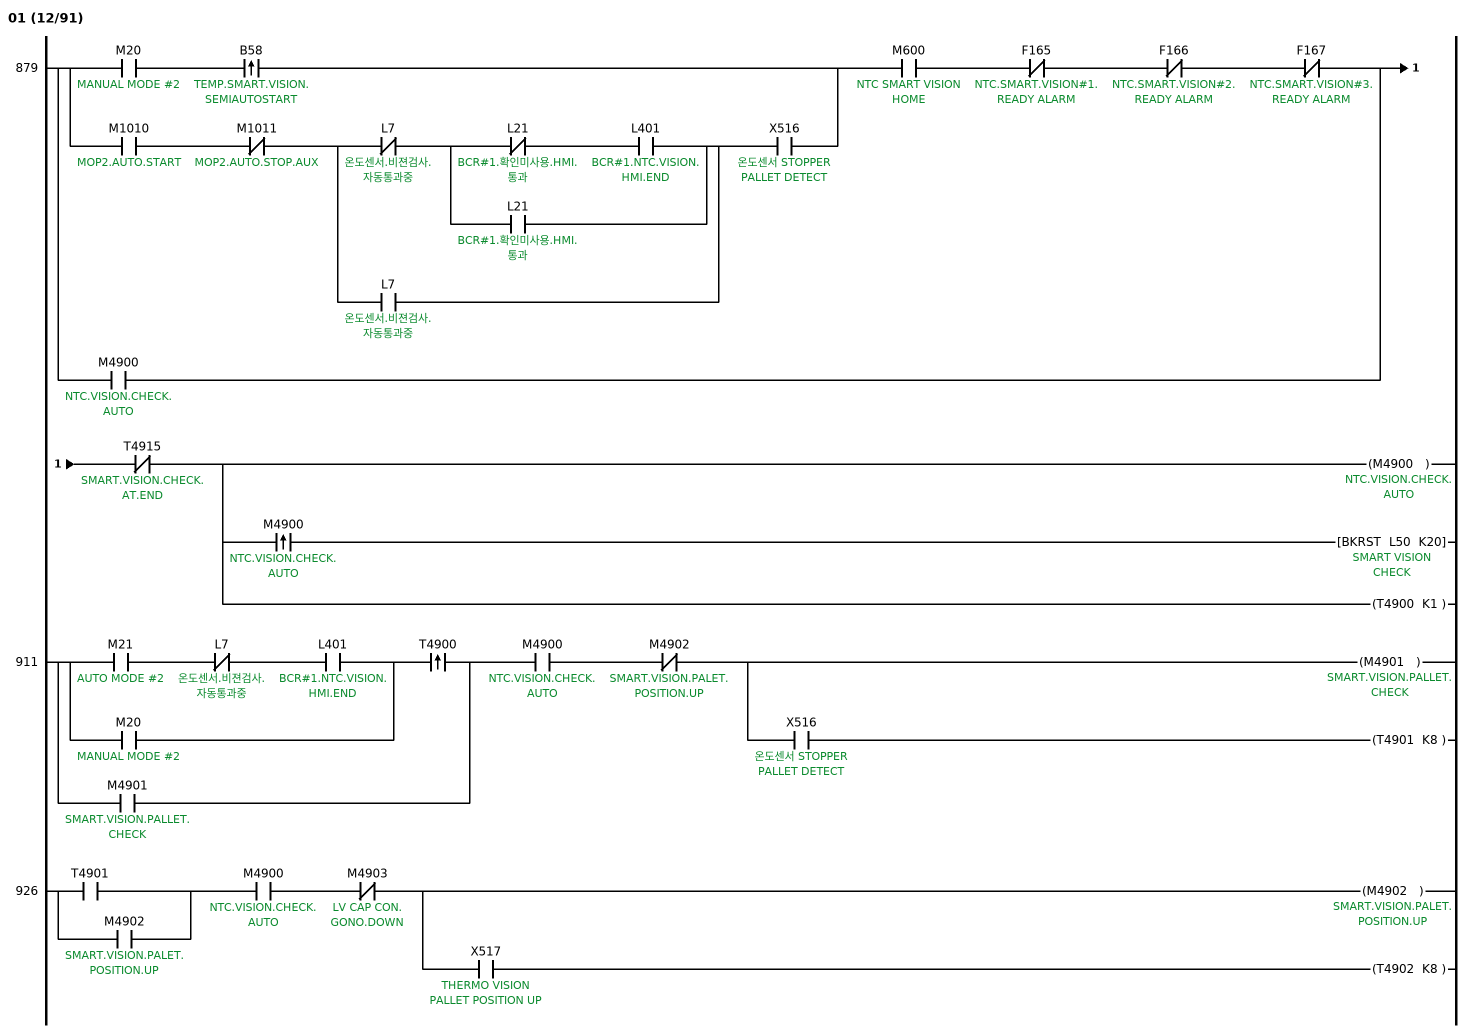
879   LD      M20  ; MANUAL MODE #2
      ANDP    B58  ; TEMP.SMART.VISION.SEMIAUTOSTART
      LD      M1010  ; MOP2.AUTO.START
      ANI     M1011  ; MOP2.AUTO.STOP.AUX
      LDI     L7  ; 온도센서.비젼검사.자동통과중
      LDI     L21  ; BCR#1.확인미사용.HMI.통과
      AND     L401  ; BCR#1.NTC.VISION.HMI.END
      OR      L21  ; BCR#1.확인미사용.HMI.통과
      ANB
      OR      L7  ; 온도센서.비젼검사.자동통과중
      ANB
      AND     X516  ; 온도센서 STOPPER PALLET DETECT
      ORB
      AND     M600  ; NTC SMART VISION HOME
      ANI     F165  ; NTC.SMART.VISION#1.READY ALARM
      ANI     F166  ; NTC.SMART.VISION#2.READY ALARM
      ANI     F167  ; NTC.SMART.VISION#3.READY ALARM
      OR      M4900  ; NTC.VISION.CHECK.AUTO
      ANI     T4915  ; SMART.VISION.CHECK.AT.END
      OUT     M4900  ; NTC.VISION.CHECK.AUTO
      MPS
      ANDP    M4900  ; NTC.VISION.CHECK.AUTO
      BKRST   L50 K20  ; SMART VISION CHECK
      MPP
      OUT     T4900 K1
911   LD      M21  ; AUTO MODE #2
      ANI     L7  ; 온도센서.비젼검사.자동통과중
      AND     L401  ; BCR#1.NTC.VISION.HMI.END
      OR      M20  ; MANUAL MODE #2
      ANDP    T4900
      OR      M4901  ; SMART.VISION.PALLET.CHECK
      AND     M4900  ; NTC.VISION.CHECK.AUTO
      ANI     M4902  ; SMART.VISION.PALET.POSITION.UP
      OUT     M4901  ; SMART.VISION.PALLET.CHECK
      AND     X516  ; 온도센서 STOPPER PALLET DETECT
      OUT     T4901 K8
926   LD      T4901
      OR      M4902  ; SMART.VISION.PALET.POSITION.UP
      AND     M4900  ; NTC.VISION.CHECK.AUTO
      ANI     M4903  ; LV CAP CON. GONO.DOWN
      OUT     M4902  ; SMART.VISION.PALET.POSITION.UP
      AND     X517  ; THERMO VISION PALLET POSITION UP
      OUT     T4902 K8
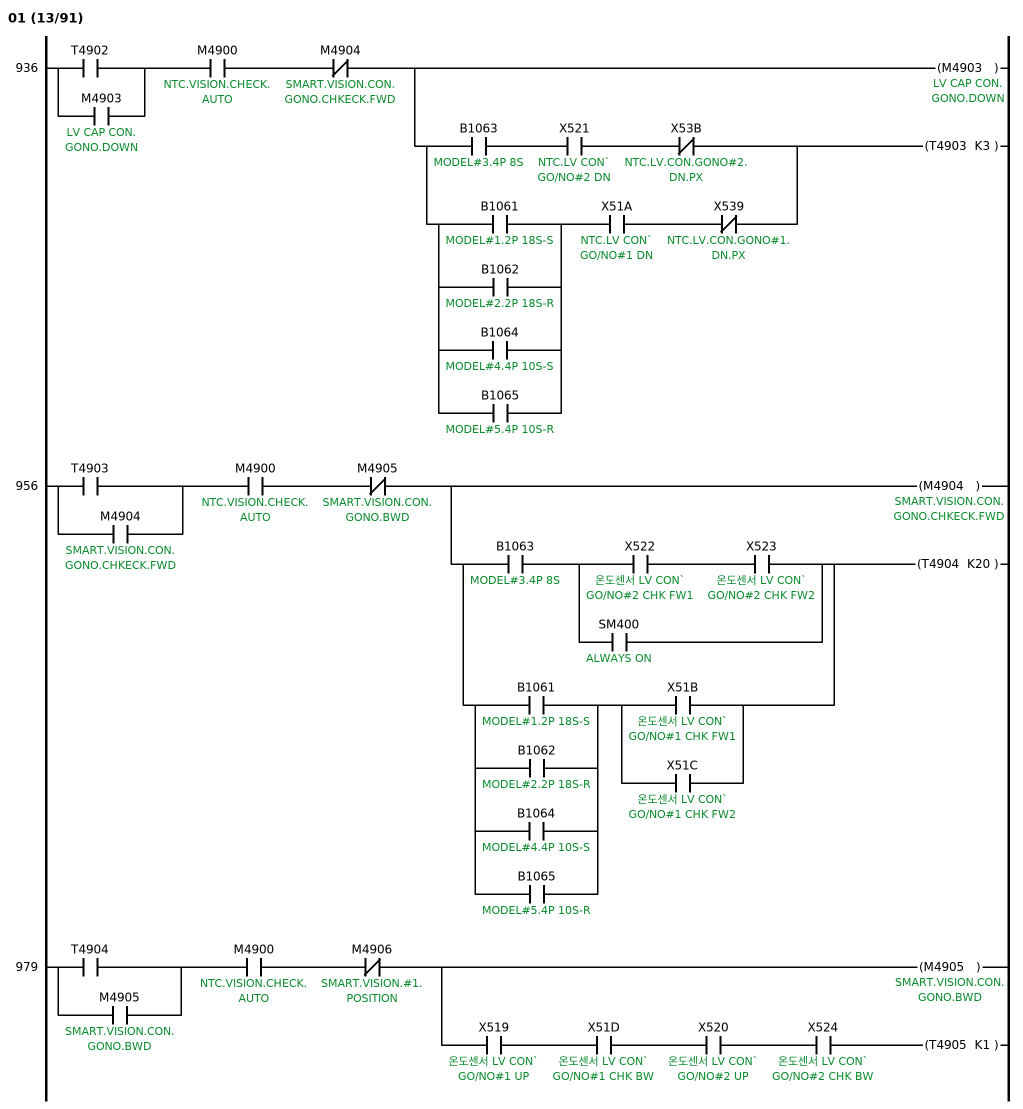
936   LD      T4902
      OR      M4903  ; LV CAP CON. GONO.DOWN
      AND     M4900  ; NTC.VISION.CHECK.AUTO
      ANI     M4904  ; SMART.VISION.CON.GONO.CHKECK.FWD
      OUT     M4903  ; LV CAP CON. GONO.DOWN
      LD      B1063  ; MODEL#3.4P 8S
      AND     X521  ; NTC.LV CON` GO/NO#2 DN
      ANI     X53B  ; NTC.LV.CON.GONO#2.DN.PX
      LD      B1061  ; MODEL#1.2P 18S-S
      OR      B1062  ; MODEL#2.2P 18S-R
      OR      B1064  ; MODEL#4.4P 10S-S
      OR      B1065  ; MODEL#5.4P 10S-R
      AND     X51A  ; NTC.LV CON` GO/NO#1 DN
      ANI     X539  ; NTC.LV.CON.GONO#1.DN.PX
      ORB
      ANB
      OUT     T4903 K3
956   LD      T4903
      OR      M4904  ; SMART.VISION.CON.GONO.CHKECK.FWD
      AND     M4900  ; NTC.VISION.CHECK.AUTO
      ANI     M4905  ; SMART.VISION.CON.GONO.BWD
      OUT     M4904  ; SMART.VISION.CON.GONO.CHKECK.FWD
      LD      B1063  ; MODEL#3.4P 8S
      LD      X522  ; 온도센서 LV CON` GO/NO#2 CHK FW1
      AND     X523  ; 온도센서 LV CON` GO/NO#2 CHK FW2
      OR      SM400  ; ALWAYS ON
      ANB
      LD      B1061  ; MODEL#1.2P 18S-S
      OR      B1062  ; MODEL#2.2P 18S-R
      OR      B1064  ; MODEL#4.4P 10S-S
      OR      B1065  ; MODEL#5.4P 10S-R
      LD      X51B  ; 온도센서 LV CON` GO/NO#1 CHK FW1
      OR      X51C  ; 온도센서 LV CON` GO/NO#1 CHK FW2
      ANB
      ORB
      ANB
      OUT     T4904 K20
979   LD      T4904
      OR      M4905  ; SMART.VISION.CON.GONO.BWD
      AND     M4900  ; NTC.VISION.CHECK.AUTO
      ANI     M4906  ; SMART.VISION.#1.POSITION
      OUT     M4905  ; SMART.VISION.CON.GONO.BWD
      AND     X519  ; 온도센서 LV CON` GO/NO#1 UP
      AND     X51D  ; 온도센서 LV CON` GO/NO#1 CHK BW
      AND     X520  ; 온도센서 LV CON` GO/NO#2 UP
      AND     X524  ; 온도센서 LV CON` GO/NO#2 CHK BW
      OUT     T4905 K1
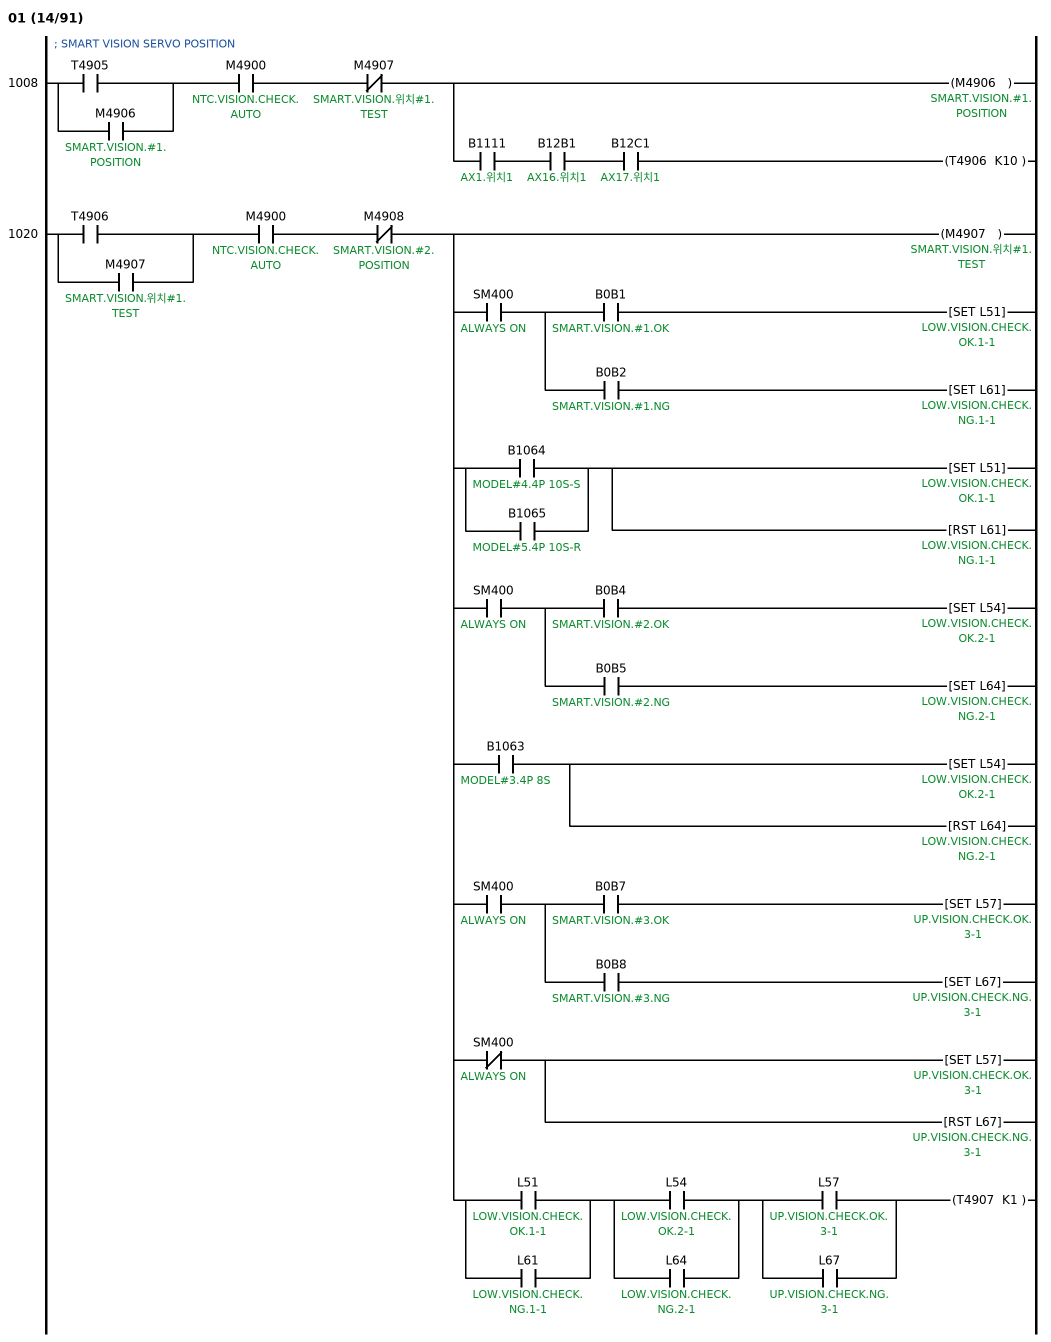
; SMART VISION SERVO POSITION
1008  LD      T4905
      OR      M4906  ; SMART.VISION.#1.POSITION
      AND     M4900  ; NTC.VISION.CHECK.AUTO
      ANI     M4907  ; SMART.VISION.위치#1.TEST
      OUT     M4906  ; SMART.VISION.#1.POSITION
      AND     B1111  ; AX1.위치1
      AND     B12B1  ; AX16.위치1
      AND     B12C1  ; AX17.위치1
      OUT     T4906 K10
1020  LD      T4906
      OR      M4907  ; SMART.VISION.위치#1.TEST
      AND     M4900  ; NTC.VISION.CHECK.AUTO
      ANI     M4908  ; SMART.VISION.#2.POSITION
      OUT     M4907  ; SMART.VISION.위치#1.TEST
      MPS
      AND     SM400  ; ALWAYS ON
      MPS
      AND     B0B1  ; SMART.VISION.#1.OK
      SET     L51  ; LOW.VISION.CHECK.OK.1-1
      MPP
      AND     B0B2  ; SMART.VISION.#1.NG
      SET     L61  ; LOW.VISION.CHECK.NG.1-1
      MRD
      LD      B1064  ; MODEL#4.4P 10S-S
      OR      B1065  ; MODEL#5.4P 10S-R
      ANB
      SET     L51  ; LOW.VISION.CHECK.OK.1-1
      RST     L61  ; LOW.VISION.CHECK.NG.1-1
      MRD
      AND     SM400  ; ALWAYS ON
      MPS
      AND     B0B4  ; SMART.VISION.#2.OK
      SET     L54  ; LOW.VISION.CHECK.OK.2-1
      MPP
      AND     B0B5  ; SMART.VISION.#2.NG
      SET     L64  ; LOW.VISION.CHECK.NG.2-1
      MRD
      AND     B1063  ; MODEL#3.4P 8S
      SET     L54  ; LOW.VISION.CHECK.OK.2-1
      RST     L64  ; LOW.VISION.CHECK.NG.2-1
      MRD
      AND     SM400  ; ALWAYS ON
      MPS
      AND     B0B7  ; SMART.VISION.#3.OK
      SET     L57  ; UP.VISION.CHECK.OK.3-1
      MPP
      AND     B0B8  ; SMART.VISION.#3.NG
      SET     L67  ; UP.VISION.CHECK.NG.3-1
      MRD
      ANI     SM400  ; ALWAYS ON
      SET     L57  ; UP.VISION.CHECK.OK.3-1
      RST     L67  ; UP.VISION.CHECK.NG.3-1
      MPP
      LD      L51  ; LOW.VISION.CHECK.OK.1-1
      OR      L61  ; LOW.VISION.CHECK.NG.1-1
      ANB
      LD      L54  ; LOW.VISION.CHECK.OK.2-1
      OR      L64  ; LOW.VISION.CHECK.NG.2-1
      ANB
      LD      L57  ; UP.VISION.CHECK.OK.3-1
      OR      L67  ; UP.VISION.CHECK.NG.3-1
      ANB
      OUT     T4907 K1
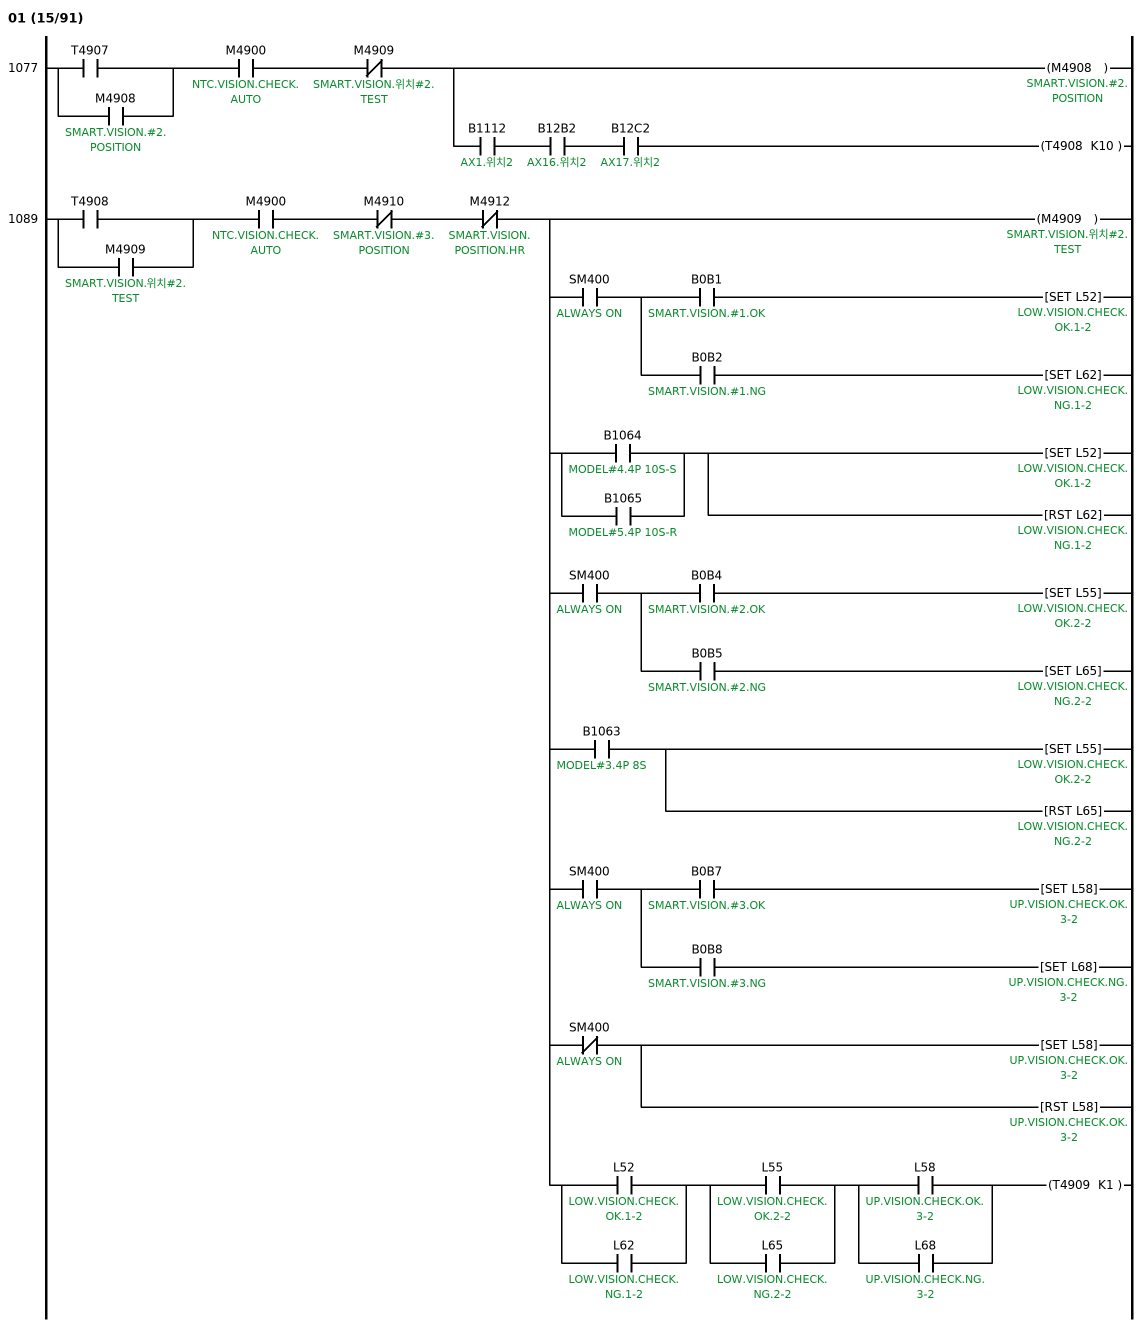
1077  LD      T4907
      OR      M4908  ; SMART.VISION.#2.POSITION
      AND     M4900  ; NTC.VISION.CHECK.AUTO
      ANI     M4909  ; SMART.VISION.위치#2.TEST
      OUT     M4908  ; SMART.VISION.#2.POSITION
      AND     B1112  ; AX1.위치2
      AND     B12B2  ; AX16.위치2
      AND     B12C2  ; AX17.위치2
      OUT     T4908 K10
1089  LD      T4908
      OR      M4909  ; SMART.VISION.위치#2.TEST
      AND     M4900  ; NTC.VISION.CHECK.AUTO
      ANI     M4910  ; SMART.VISION.#3.POSITION
      ANI     M4912  ; SMART.VISION.POSITION.HR
      OUT     M4909  ; SMART.VISION.위치#2.TEST
      MPS
      AND     SM400  ; ALWAYS ON
      MPS
      AND     B0B1  ; SMART.VISION.#1.OK
      SET     L52  ; LOW.VISION.CHECK.OK.1-2
      MPP
      AND     B0B2  ; SMART.VISION.#1.NG
      SET     L62  ; LOW.VISION.CHECK.NG.1-2
      MRD
      LD      B1064  ; MODEL#4.4P 10S-S
      OR      B1065  ; MODEL#5.4P 10S-R
      ANB
      SET     L52  ; LOW.VISION.CHECK.OK.1-2
      RST     L62  ; LOW.VISION.CHECK.NG.1-2
      MRD
      AND     SM400  ; ALWAYS ON
      MPS
      AND     B0B4  ; SMART.VISION.#2.OK
      SET     L55  ; LOW.VISION.CHECK.OK.2-2
      MPP
      AND     B0B5  ; SMART.VISION.#2.NG
      SET     L65  ; LOW.VISION.CHECK.NG.2-2
      MRD
      AND     B1063  ; MODEL#3.4P 8S
      SET     L55  ; LOW.VISION.CHECK.OK.2-2
      RST     L65  ; LOW.VISION.CHECK.NG.2-2
      MRD
      AND     SM400  ; ALWAYS ON
      MPS
      AND     B0B7  ; SMART.VISION.#3.OK
      SET     L58  ; UP.VISION.CHECK.OK.3-2
      MPP
      AND     B0B8  ; SMART.VISION.#3.NG
      SET     L68  ; UP.VISION.CHECK.NG.3-2
      MRD
      ANI     SM400  ; ALWAYS ON
      SET     L58  ; UP.VISION.CHECK.OK.3-2
      RST     L58  ; UP.VISION.CHECK.OK.3-2
      MPP
      LD      L52  ; LOW.VISION.CHECK.OK.1-2
      OR      L62  ; LOW.VISION.CHECK.NG.1-2
      ANB
      LD      L55  ; LOW.VISION.CHECK.OK.2-2
      OR      L65  ; LOW.VISION.CHECK.NG.2-2
      ANB
      LD      L58  ; UP.VISION.CHECK.OK.3-2
      OR      L68  ; UP.VISION.CHECK.NG.3-2
      ANB
      OUT     T4909 K1
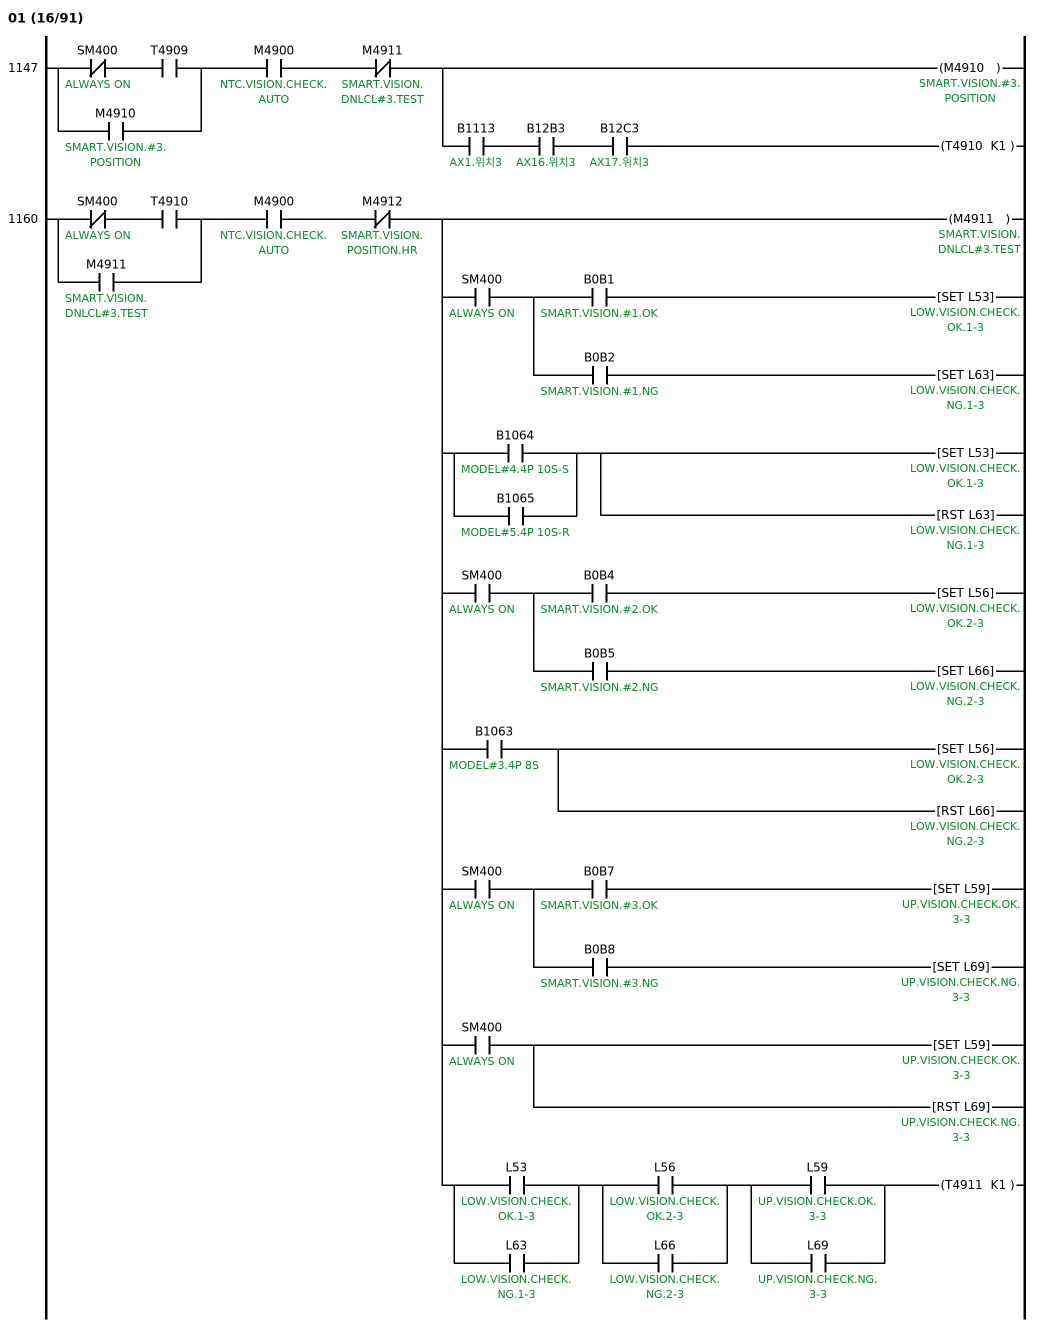
1147  LDI     SM400  ; ALWAYS ON
      AND     T4909
      OR      M4910  ; SMART.VISION.#3.POSITION
      AND     M4900  ; NTC.VISION.CHECK.AUTO
      ANI     M4911  ; SMART.VISION.DNLCL#3.TEST
      OUT     M4910  ; SMART.VISION.#3.POSITION
      AND     B1113  ; AX1.위치3
      AND     B12B3  ; AX16.위치3
      AND     B12C3  ; AX17.위치3
      OUT     T4910 K1
1160  LDI     SM400  ; ALWAYS ON
      AND     T4910
      OR      M4911  ; SMART.VISION.DNLCL#3.TEST
      AND     M4900  ; NTC.VISION.CHECK.AUTO
      ANI     M4912  ; SMART.VISION.POSITION.HR
      OUT     M4911  ; SMART.VISION.DNLCL#3.TEST
      MPS
      AND     SM400  ; ALWAYS ON
      MPS
      AND     B0B1  ; SMART.VISION.#1.OK
      SET     L53  ; LOW.VISION.CHECK.OK.1-3
      MPP
      AND     B0B2  ; SMART.VISION.#1.NG
      SET     L63  ; LOW.VISION.CHECK.NG.1-3
      MRD
      LD      B1064  ; MODEL#4.4P 10S-S
      OR      B1065  ; MODEL#5.4P 10S-R
      ANB
      SET     L53  ; LOW.VISION.CHECK.OK.1-3
      RST     L63  ; LOW.VISION.CHECK.NG.1-3
      MRD
      AND     SM400  ; ALWAYS ON
      MPS
      AND     B0B4  ; SMART.VISION.#2.OK
      SET     L56  ; LOW.VISION.CHECK.OK.2-3
      MPP
      AND     B0B5  ; SMART.VISION.#2.NG
      SET     L66  ; LOW.VISION.CHECK.NG.2-3
      MRD
      AND     B1063  ; MODEL#3.4P 8S
      SET     L56  ; LOW.VISION.CHECK.OK.2-3
      RST     L66  ; LOW.VISION.CHECK.NG.2-3
      MRD
      AND     SM400  ; ALWAYS ON
      MPS
      AND     B0B7  ; SMART.VISION.#3.OK
      SET     L59  ; UP.VISION.CHECK.OK.3-3
      MPP
      AND     B0B8  ; SMART.VISION.#3.NG
      SET     L69  ; UP.VISION.CHECK.NG.3-3
      MRD
      AND     SM400  ; ALWAYS ON
      SET     L59  ; UP.VISION.CHECK.OK.3-3
      RST     L69  ; UP.VISION.CHECK.NG.3-3
      MPP
      LD      L53  ; LOW.VISION.CHECK.OK.1-3
      OR      L63  ; LOW.VISION.CHECK.NG.1-3
      ANB
      LD      L56  ; LOW.VISION.CHECK.OK.2-3
      OR      L66  ; LOW.VISION.CHECK.NG.2-3
      ANB
      LD      L59  ; UP.VISION.CHECK.OK.3-3
      OR      L69  ; UP.VISION.CHECK.NG.3-3
      ANB
      OUT     T4911 K1
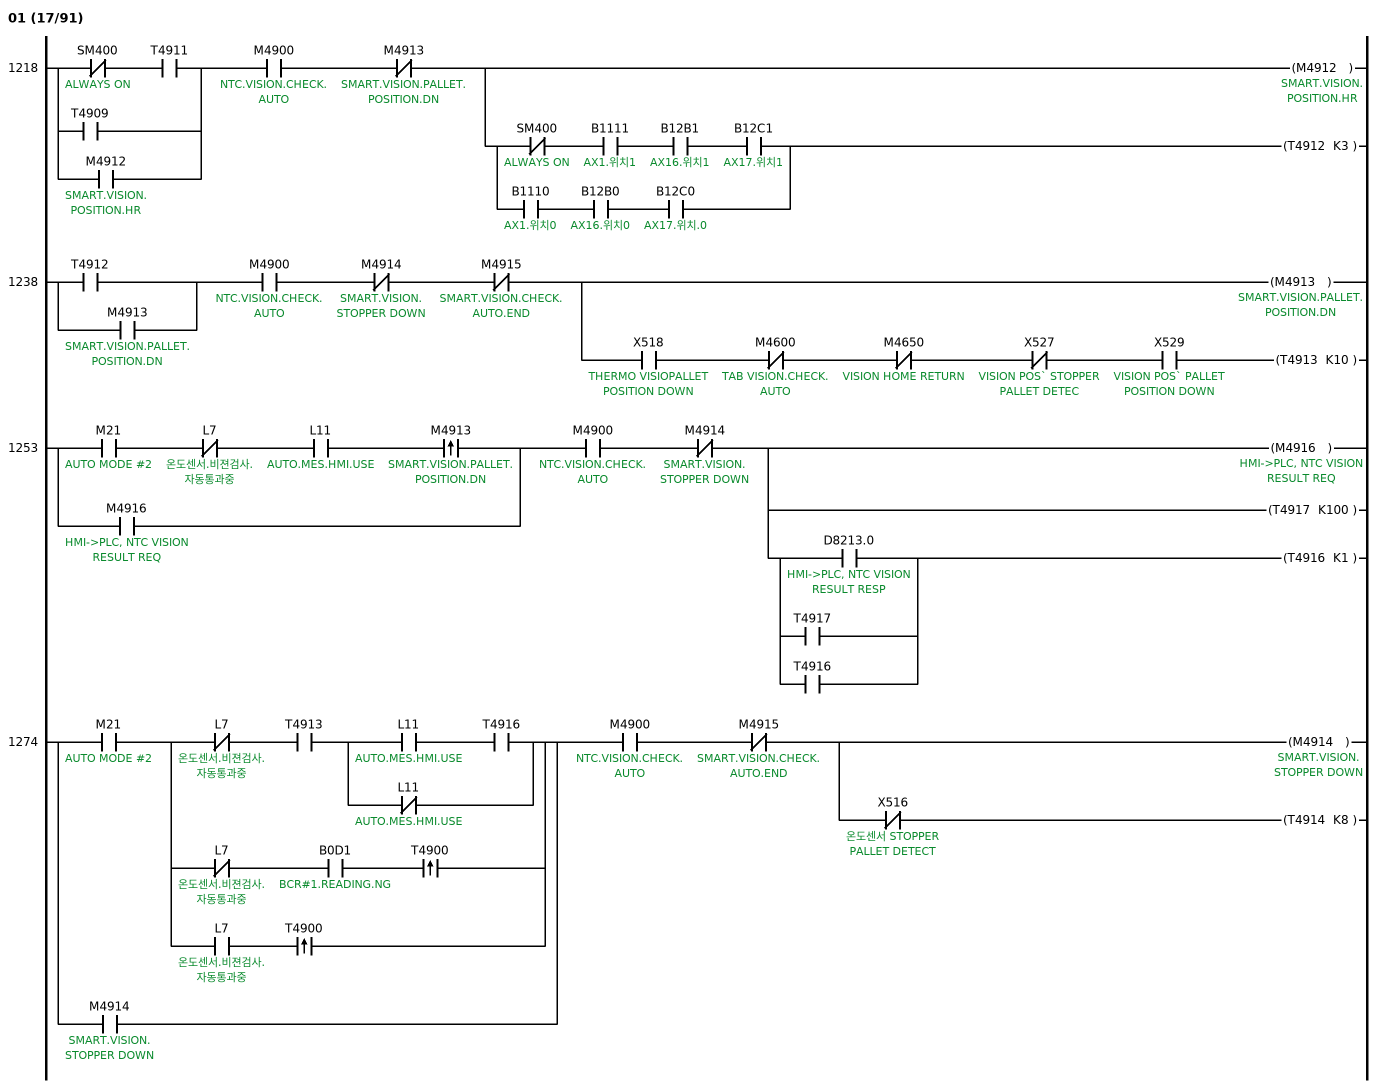
1218  LDI     SM400  ; ALWAYS ON
      AND     T4911
      OR      T4909
      OR      M4912  ; SMART.VISION.POSITION.HR
      AND     M4900  ; NTC.VISION.CHECK.AUTO
      ANI     M4913  ; SMART.VISION.PALLET.POSITION.DN
      OUT     M4912  ; SMART.VISION.POSITION.HR
      LDI     SM400  ; ALWAYS ON
      AND     B1111  ; AX1.위치1
      AND     B12B1  ; AX16.위치1
      AND     B12C1  ; AX17.위치1
      LD      B1110  ; AX1.위치0
      AND     B12B0  ; AX16.위치0
      AND     B12C0  ; AX17.위치.0
      ORB
      ANB
      OUT     T4912 K3
1238  LD      T4912
      OR      M4913  ; SMART.VISION.PALLET.POSITION.DN
      AND     M4900  ; NTC.VISION.CHECK.AUTO
      ANI     M4914  ; SMART.VISION.STOPPER DOWN
      ANI     M4915  ; SMART.VISION.CHECK.AUTO.END
      OUT     M4913  ; SMART.VISION.PALLET.POSITION.DN
      AND     X518  ; THERMO VISIOPALLET POSITION DOWN
      ANI     M4600  ; TAB VISION.CHECK.AUTO
      ANI     M4650  ; VISION HOME RETURN
      ANI     X527  ; VISION POS` STOPPER PALLET DETEC
      AND     X529  ; VISION POS` PALLET POSITION DOWN
      OUT     T4913 K10
1253  LD      M21  ; AUTO MODE #2
      ANI     L7  ; 온도센서.비젼검사.자동통과중
      AND     L11  ; AUTO.MES.HMI.USE
      ANDP    M4913  ; SMART.VISION.PALLET.POSITION.DN
      OR      M4916  ; HMI->PLC, NTC VISION RESULT REQ
      AND     M4900  ; NTC.VISION.CHECK.AUTO
      ANI     M4914  ; SMART.VISION.STOPPER DOWN
      OUT     M4916  ; HMI->PLC, NTC VISION RESULT REQ
      OUT     T4917 K100
      LD      D8213.0  ; HMI->PLC, NTC VISION RESULT RESP
      OR      T4917
      OR      T4916
      ANB
      OUT     T4916 K1
1274  LD      M21  ; AUTO MODE #2
      LDI     L7  ; 온도센서.비젼검사.자동통과중
      AND     T4913
      LD      L11  ; AUTO.MES.HMI.USE
      AND     T4916
      ORI     L11  ; AUTO.MES.HMI.USE
      ANB
      LDI     L7  ; 온도센서.비젼검사.자동통과중
      AND     B0D1  ; BCR#1.READING.NG
      ANDP    T4900
      ORB
      LD      L7  ; 온도센서.비젼검사.자동통과중
      ANDP    T4900
      ORB
      ANB
      OR      M4914  ; SMART.VISION.STOPPER DOWN
      AND     M4900  ; NTC.VISION.CHECK.AUTO
      ANI     M4915  ; SMART.VISION.CHECK.AUTO.END
      OUT     M4914  ; SMART.VISION.STOPPER DOWN
      ANI     X516  ; 온도센서 STOPPER PALLET DETECT
      OUT     T4914 K8
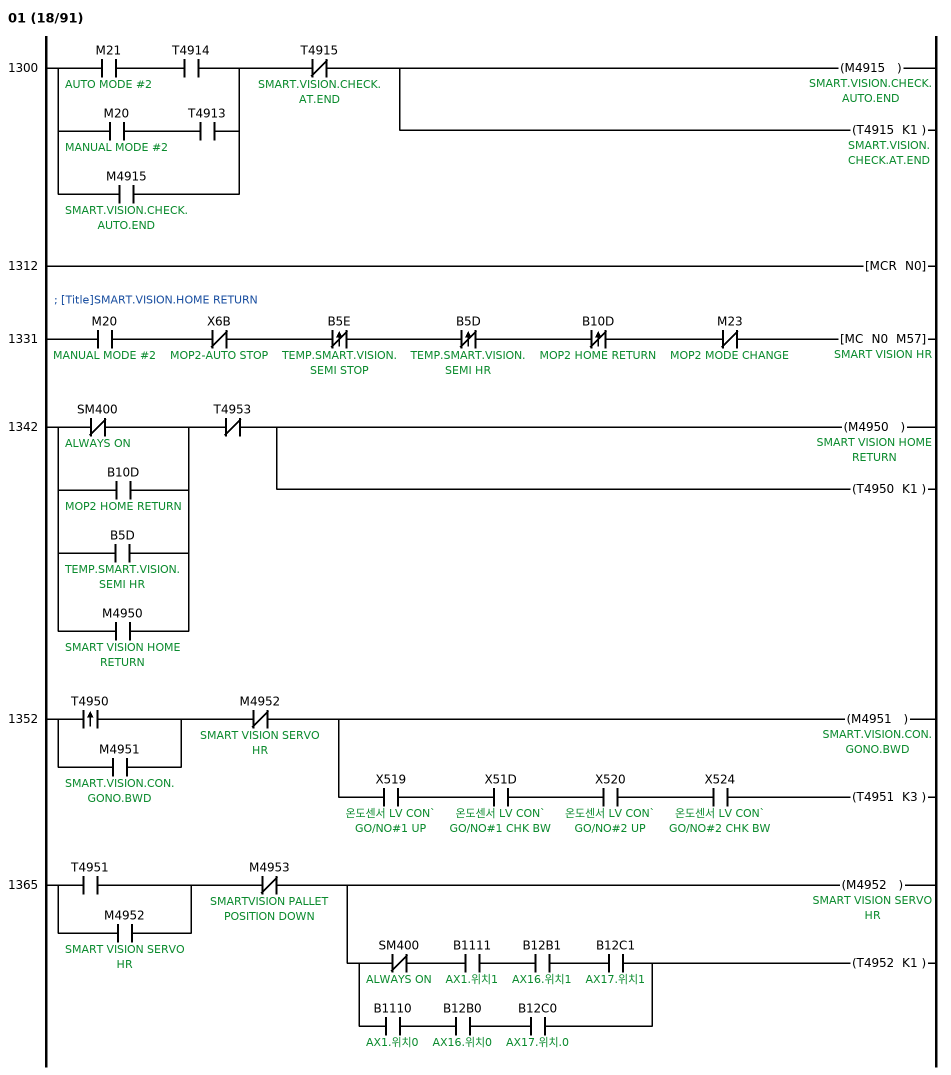
1300  LD      M21  ; AUTO MODE #2
      AND     T4914
      LD      M20  ; MANUAL MODE #2
      AND     T4913
      ORB
      OR      M4915  ; SMART.VISION.CHECK.AUTO.END
      ANI     T4915  ; SMART.VISION.CHECK.AT.END
      OUT     M4915  ; SMART.VISION.CHECK.AUTO.END
      OUT     T4915 K1  ; SMART.VISION.CHECK.AT.END
1312  MCR     N0
; [Title]SMART.VISION.HOME RETURN
1331  LD      M20  ; MANUAL MODE #2
      ANI     X6B  ; MOP2-AUTO STOP
      ANDPI   B5E  ; TEMP.SMART.VISION.SEMI STOP
      ANDPI   B5D  ; TEMP.SMART.VISION.SEMI HR
      ANDPI   B10D  ; MOP2 HOME RETURN
      ANI     M23  ; MOP2 MODE CHANGE
      MC      N0 M57  ; SMART VISION HR
1342  LDI     SM400  ; ALWAYS ON
      OR      B10D  ; MOP2 HOME RETURN
      OR      B5D  ; TEMP.SMART.VISION.SEMI HR
      OR      M4950  ; SMART VISION HOME RETURN
      ANI     T4953
      OUT     M4950  ; SMART VISION HOME RETURN
      OUT     T4950 K1
1352  LDP     T4950
      OR      M4951  ; SMART.VISION.CON.GONO.BWD
      ANI     M4952  ; SMART VISION SERVO HR
      OUT     M4951  ; SMART.VISION.CON.GONO.BWD
      AND     X519  ; 온도센서 LV CON` GO/NO#1 UP
      AND     X51D  ; 온도센서 LV CON` GO/NO#1 CHK BW
      AND     X520  ; 온도센서 LV CON` GO/NO#2 UP
      AND     X524  ; 온도센서 LV CON` GO/NO#2 CHK BW
      OUT     T4951 K3
1365  LD      T4951
      OR      M4952  ; SMART VISION SERVO HR
      ANI     M4953  ; SMARTVISION PALLET POSITION DOWN
      OUT     M4952  ; SMART VISION SERVO HR
      LDI     SM400  ; ALWAYS ON
      AND     B1111  ; AX1.위치1
      AND     B12B1  ; AX16.위치1
      AND     B12C1  ; AX17.위치1
      LD      B1110  ; AX1.위치0
      AND     B12B0  ; AX16.위치0
      AND     B12C0  ; AX17.위치.0
      ORB
      ANB
      OUT     T4952 K1
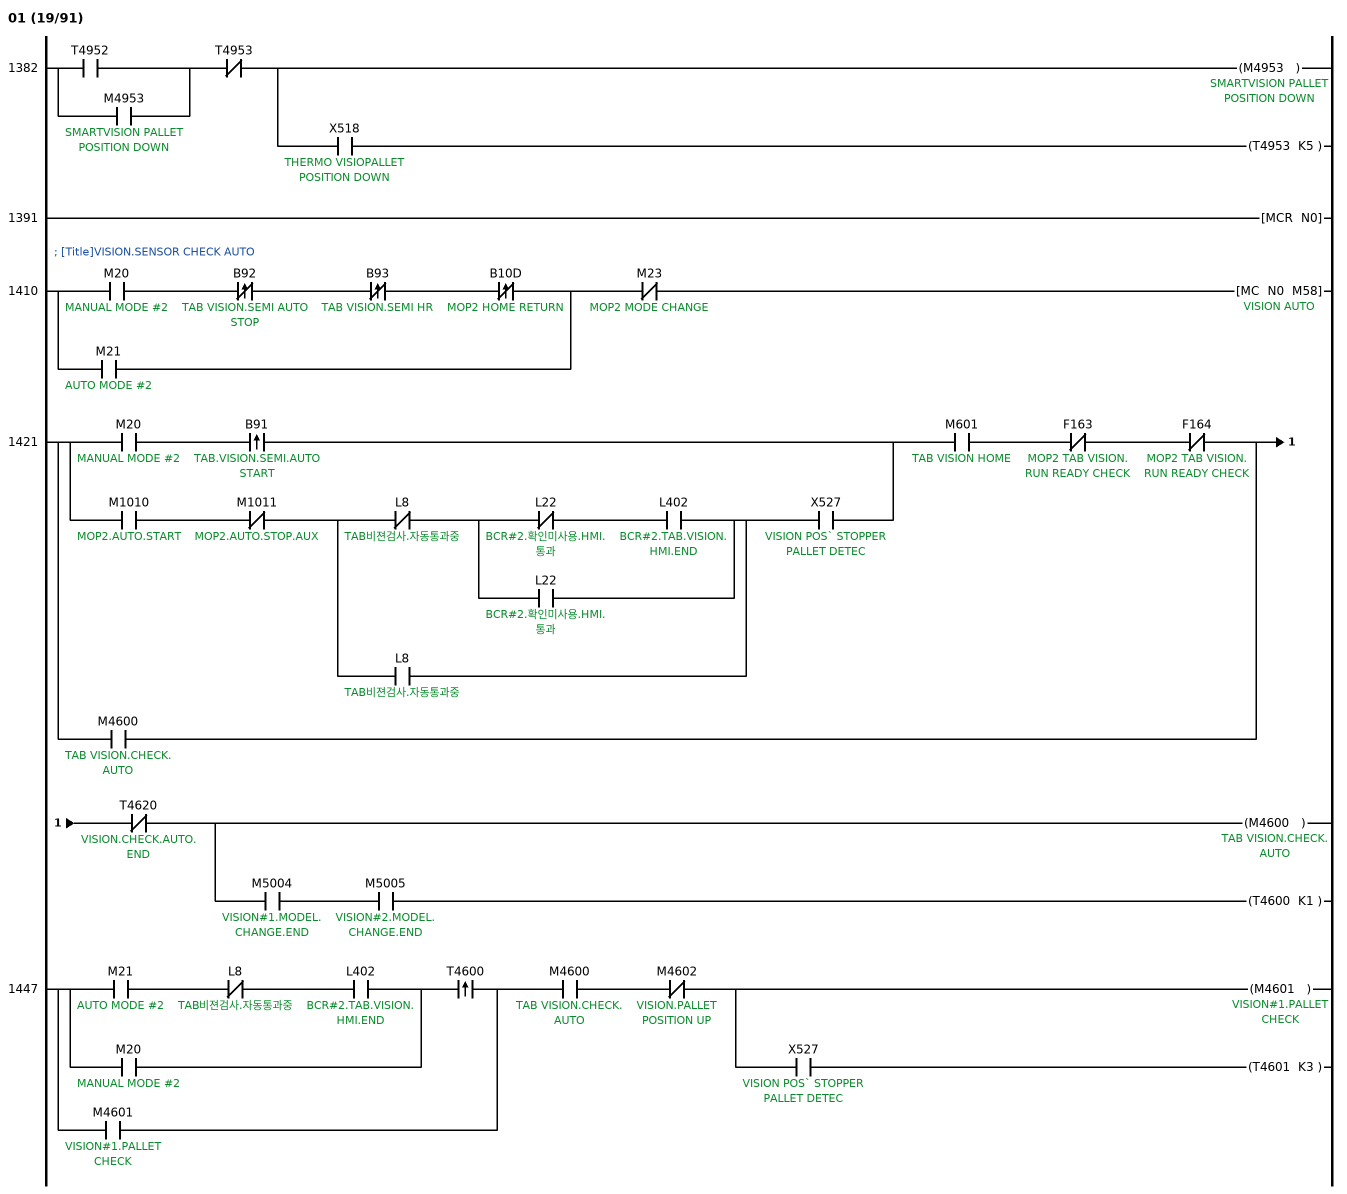
1382  LD      T4952
      OR      M4953  ; SMARTVISION PALLET POSITION DOWN
      ANI     T4953
      OUT     M4953  ; SMARTVISION PALLET POSITION DOWN
      AND     X518  ; THERMO VISIOPALLET POSITION DOWN
      OUT     T4953 K5
1391  MCR     N0
; [Title]VISION.SENSOR CHECK AUTO
1410  LD      M20  ; MANUAL MODE #2
      ANDPI   B92  ; TAB VISION.SEMI AUTO STOP
      ANDPI   B93  ; TAB VISION.SEMI HR
      ANDPI   B10D  ; MOP2 HOME RETURN
      OR      M21  ; AUTO MODE #2
      ANI     M23  ; MOP2 MODE CHANGE
      MC      N0 M58  ; VISION AUTO
1421  LD      M20  ; MANUAL MODE #2
      ANDP    B91  ; TAB.VISION.SEMI.AUTO START
      LD      M1010  ; MOP2.AUTO.START
      ANI     M1011  ; MOP2.AUTO.STOP.AUX
      LDI     L8  ; TAB비젼검사.자동통과중
      LDI     L22  ; BCR#2.확인미사용.HMI.통과
      AND     L402  ; BCR#2.TAB.VISION.HMI.END
      OR      L22  ; BCR#2.확인미사용.HMI.통과
      ANB
      OR      L8  ; TAB비젼검사.자동통과중
      ANB
      AND     X527  ; VISION POS` STOPPER PALLET DETEC
      ORB
      AND     M601  ; TAB VISION HOME
      ANI     F163  ; MOP2 TAB VISION. RUN READY CHECK
      ANI     F164  ; MOP2 TAB VISION. RUN READY CHECK
      OR      M4600  ; TAB VISION.CHECK.AUTO
      ANI     T4620  ; VISION.CHECK.AUTO.END
      OUT     M4600  ; TAB VISION.CHECK.AUTO
      AND     M5004  ; VISION#1.MODEL.CHANGE.END
      AND     M5005  ; VISION#2.MODEL.CHANGE.END
      OUT     T4600 K1
1447  LD      M21  ; AUTO MODE #2
      ANI     L8  ; TAB비젼검사.자동통과중
      AND     L402  ; BCR#2.TAB.VISION.HMI.END
      OR      M20  ; MANUAL MODE #2
      ANDP    T4600
      OR      M4601  ; VISION#1.PALLET CHECK
      AND     M4600  ; TAB VISION.CHECK.AUTO
      ANI     M4602  ; VISION.PALLET POSITION UP
      OUT     M4601  ; VISION#1.PALLET CHECK
      AND     X527  ; VISION POS` STOPPER PALLET DETEC
      OUT     T4601 K3
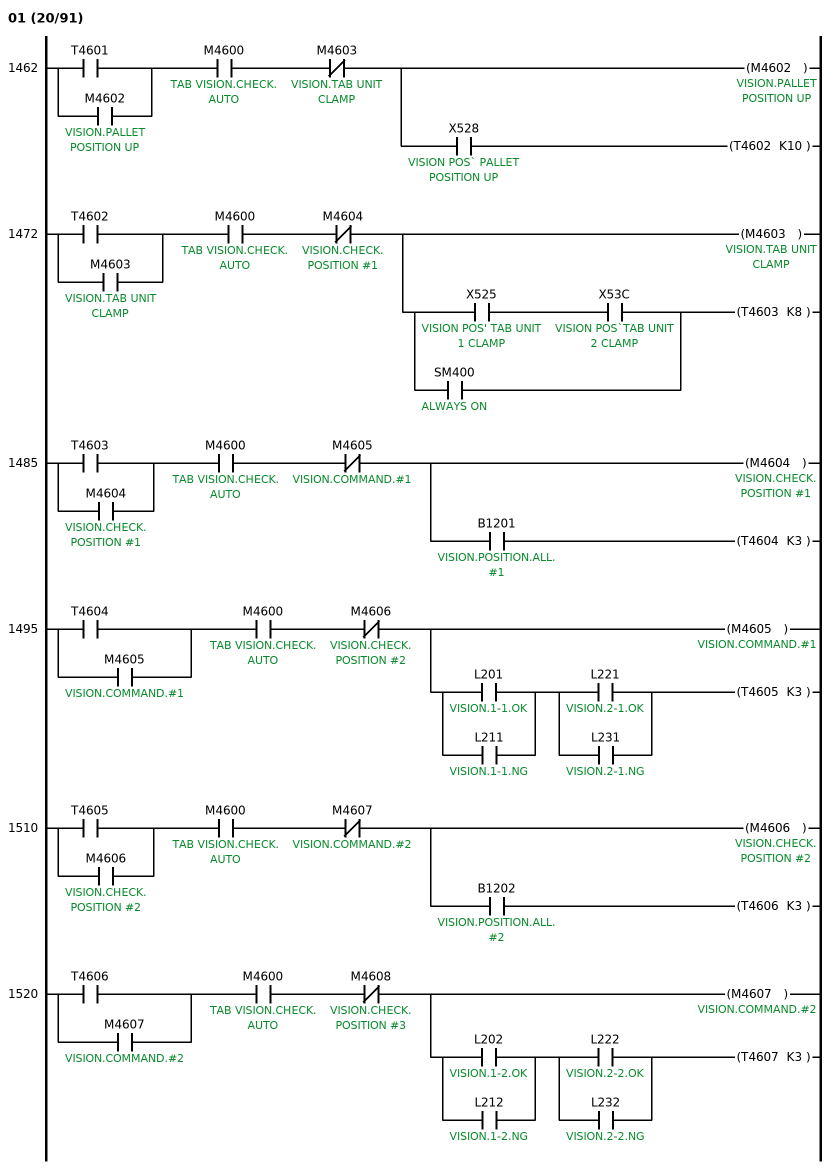
1462  LD      T4601
      OR      M4602  ; VISION.PALLET POSITION UP
      AND     M4600  ; TAB VISION.CHECK.AUTO
      ANI     M4603  ; VISION.TAB UNIT CLAMP
      OUT     M4602  ; VISION.PALLET POSITION UP
      AND     X528  ; VISION POS` PALLET POSITION UP
      OUT     T4602 K10
1472  LD      T4602
      OR      M4603  ; VISION.TAB UNIT CLAMP
      AND     M4600  ; TAB VISION.CHECK.AUTO
      ANI     M4604  ; VISION.CHECK.POSITION #1
      OUT     M4603  ; VISION.TAB UNIT CLAMP
      LD      X525  ; VISION POS' TAB UNIT 1 CLAMP
      AND     X53C  ; VISION POS`TAB UNIT 2 CLAMP
      OR      SM400  ; ALWAYS ON
      ANB
      OUT     T4603 K8
1485  LD      T4603
      OR      M4604  ; VISION.CHECK.POSITION #1
      AND     M4600  ; TAB VISION.CHECK.AUTO
      ANI     M4605  ; VISION.COMMAND.#1
      OUT     M4604  ; VISION.CHECK.POSITION #1
      AND     B1201  ; VISION.POSITION.ALL.#1
      OUT     T4604 K3
1495  LD      T4604
      OR      M4605  ; VISION.COMMAND.#1
      AND     M4600  ; TAB VISION.CHECK.AUTO
      ANI     M4606  ; VISION.CHECK.POSITION #2
      OUT     M4605  ; VISION.COMMAND.#1
      LD      L201  ; VISION.1-1.OK
      OR      L211  ; VISION.1-1.NG
      ANB
      LD      L221  ; VISION.2-1.OK
      OR      L231  ; VISION.2-1.NG
      ANB
      OUT     T4605 K3
1510  LD      T4605
      OR      M4606  ; VISION.CHECK.POSITION #2
      AND     M4600  ; TAB VISION.CHECK.AUTO
      ANI     M4607  ; VISION.COMMAND.#2
      OUT     M4606  ; VISION.CHECK.POSITION #2
      AND     B1202  ; VISION.POSITION.ALL.#2
      OUT     T4606 K3
1520  LD      T4606
      OR      M4607  ; VISION.COMMAND.#2
      AND     M4600  ; TAB VISION.CHECK.AUTO
      ANI     M4608  ; VISION.CHECK.POSITION #3
      OUT     M4607  ; VISION.COMMAND.#2
      LD      L202  ; VISION.1-2.OK
      OR      L212  ; VISION.1-2.NG
      ANB
      LD      L222  ; VISION.2-2.OK
      OR      L232  ; VISION.2-2.NG
      ANB
      OUT     T4607 K3
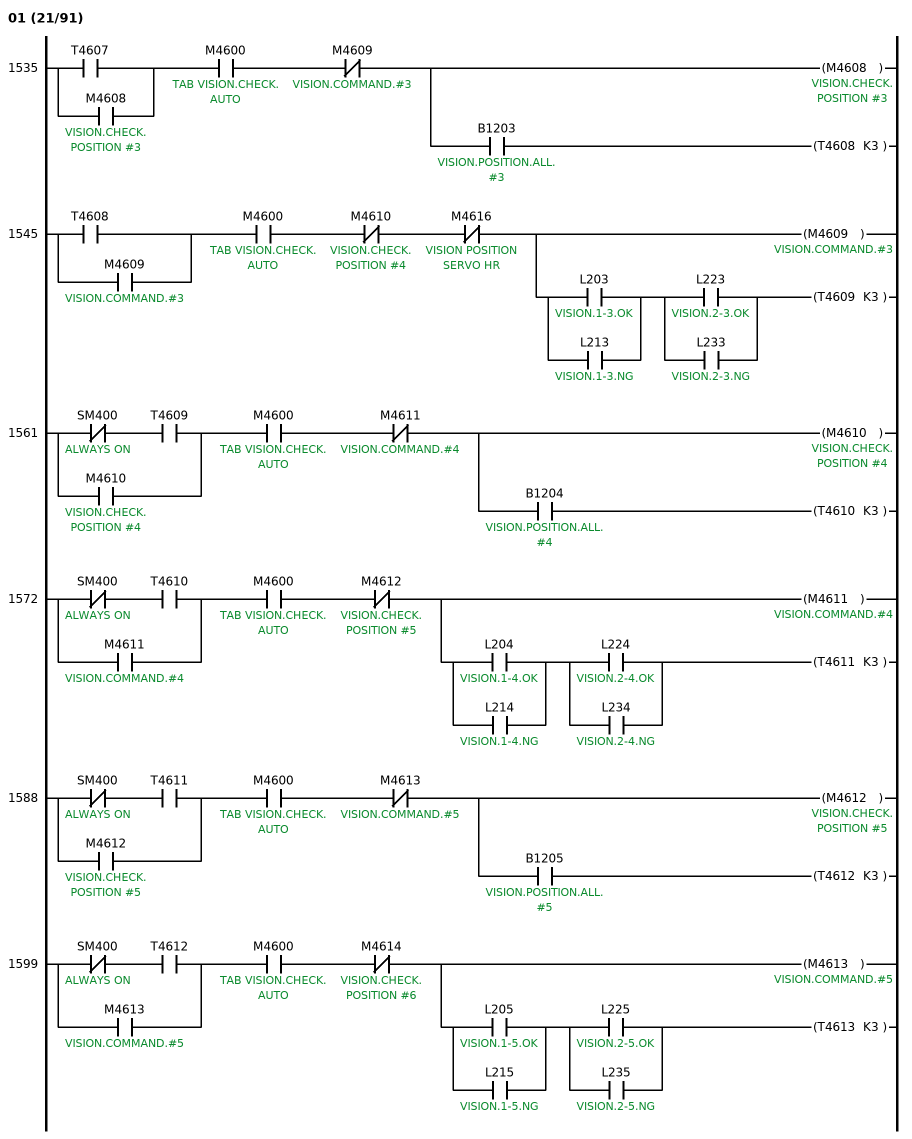
1535  LD      T4607
      OR      M4608  ; VISION.CHECK.POSITION #3
      AND     M4600  ; TAB VISION.CHECK.AUTO
      ANI     M4609  ; VISION.COMMAND.#3
      OUT     M4608  ; VISION.CHECK.POSITION #3
      AND     B1203  ; VISION.POSITION.ALL.#3
      OUT     T4608 K3
1545  LD      T4608
      OR      M4609  ; VISION.COMMAND.#3
      AND     M4600  ; TAB VISION.CHECK.AUTO
      ANI     M4610  ; VISION.CHECK.POSITION #4
      ANI     M4616  ; VISION POSITION SERVO HR
      OUT     M4609  ; VISION.COMMAND.#3
      LD      L203  ; VISION.1-3.OK
      OR      L213  ; VISION.1-3.NG
      ANB
      LD      L223  ; VISION.2-3.OK
      OR      L233  ; VISION.2-3.NG
      ANB
      OUT     T4609 K3
1561  LDI     SM400  ; ALWAYS ON
      AND     T4609
      OR      M4610  ; VISION.CHECK.POSITION #4
      AND     M4600  ; TAB VISION.CHECK.AUTO
      ANI     M4611  ; VISION.COMMAND.#4
      OUT     M4610  ; VISION.CHECK.POSITION #4
      AND     B1204  ; VISION.POSITION.ALL.#4
      OUT     T4610 K3
1572  LDI     SM400  ; ALWAYS ON
      AND     T4610
      OR      M4611  ; VISION.COMMAND.#4
      AND     M4600  ; TAB VISION.CHECK.AUTO
      ANI     M4612  ; VISION.CHECK.POSITION #5
      OUT     M4611  ; VISION.COMMAND.#4
      LD      L204  ; VISION.1-4.OK
      OR      L214  ; VISION.1-4.NG
      ANB
      LD      L224  ; VISION.2-4.OK
      OR      L234  ; VISION.2-4.NG
      ANB
      OUT     T4611 K3
1588  LDI     SM400  ; ALWAYS ON
      AND     T4611
      OR      M4612  ; VISION.CHECK.POSITION #5
      AND     M4600  ; TAB VISION.CHECK.AUTO
      ANI     M4613  ; VISION.COMMAND.#5
      OUT     M4612  ; VISION.CHECK.POSITION #5
      AND     B1205  ; VISION.POSITION.ALL.#5
      OUT     T4612 K3
1599  LDI     SM400  ; ALWAYS ON
      AND     T4612
      OR      M4613  ; VISION.COMMAND.#5
      AND     M4600  ; TAB VISION.CHECK.AUTO
      ANI     M4614  ; VISION.CHECK.POSITION #6
      OUT     M4613  ; VISION.COMMAND.#5
      LD      L205  ; VISION.1-5.OK
      OR      L215  ; VISION.1-5.NG
      ANB
      LD      L225  ; VISION.2-5.OK
      OR      L235  ; VISION.2-5.NG
      ANB
      OUT     T4613 K3
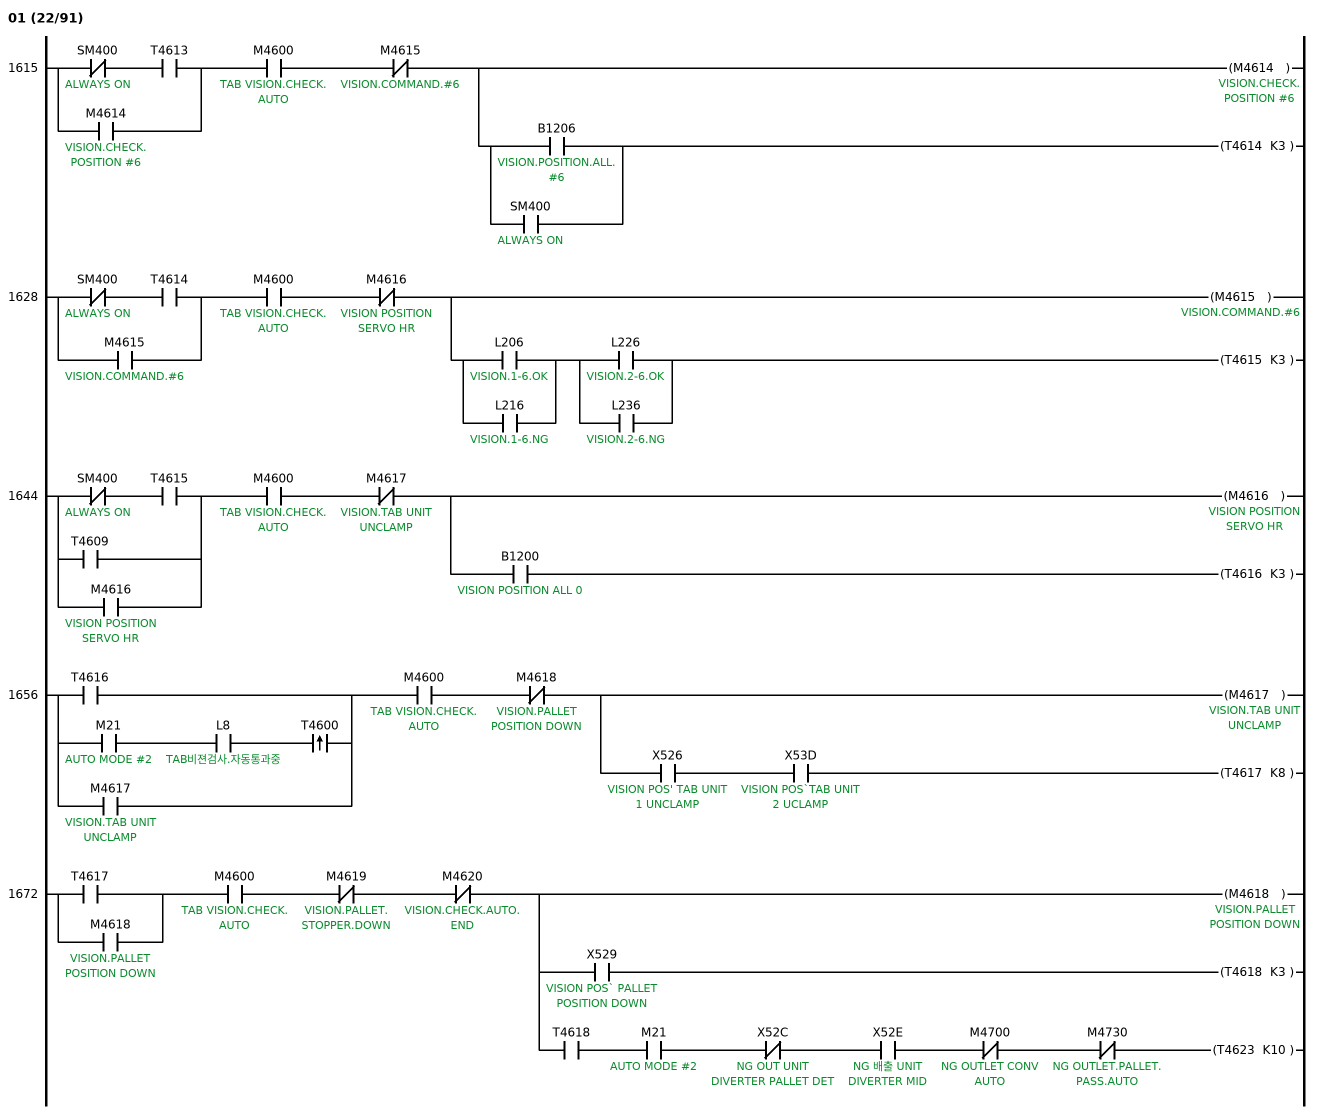
1615  LDI     SM400  ; ALWAYS ON
      AND     T4613
      OR      M4614  ; VISION.CHECK.POSITION #6
      AND     M4600  ; TAB VISION.CHECK.AUTO
      ANI     M4615  ; VISION.COMMAND.#6
      OUT     M4614  ; VISION.CHECK.POSITION #6
      LD      B1206  ; VISION.POSITION.ALL.#6
      OR      SM400  ; ALWAYS ON
      ANB
      OUT     T4614 K3
1628  LDI     SM400  ; ALWAYS ON
      AND     T4614
      OR      M4615  ; VISION.COMMAND.#6
      AND     M4600  ; TAB VISION.CHECK.AUTO
      ANI     M4616  ; VISION POSITION SERVO HR
      OUT     M4615  ; VISION.COMMAND.#6
      LD      L206  ; VISION.1-6.OK
      OR      L216  ; VISION.1-6.NG
      ANB
      LD      L226  ; VISION.2-6.OK
      OR      L236  ; VISION.2-6.NG
      ANB
      OUT     T4615 K3
1644  LDI     SM400  ; ALWAYS ON
      AND     T4615
      OR      T4609
      OR      M4616  ; VISION POSITION SERVO HR
      AND     M4600  ; TAB VISION.CHECK.AUTO
      ANI     M4617  ; VISION.TAB UNIT UNCLAMP
      OUT     M4616  ; VISION POSITION SERVO HR
      AND     B1200  ; VISION POSITION ALL 0
      OUT     T4616 K3
1656  LD      T4616
      LD      M21  ; AUTO MODE #2
      AND     L8  ; TAB비젼검사.자동통과중
      ANDP    T4600
      ORB
      OR      M4617  ; VISION.TAB UNIT UNCLAMP
      AND     M4600  ; TAB VISION.CHECK.AUTO
      ANI     M4618  ; VISION.PALLET POSITION DOWN
      OUT     M4617  ; VISION.TAB UNIT UNCLAMP
      AND     X526  ; VISION POS' TAB UNIT 1 UNCLAMP
      AND     X53D  ; VISION POS`TAB UNIT 2 UCLAMP
      OUT     T4617 K8
1672  LD      T4617
      OR      M4618  ; VISION.PALLET POSITION DOWN
      AND     M4600  ; TAB VISION.CHECK.AUTO
      ANI     M4619  ; VISION.PALLET.STOPPER.DOWN
      ANI     M4620  ; VISION.CHECK.AUTO.END
      OUT     M4618  ; VISION.PALLET POSITION DOWN
      MPS
      AND     X529  ; VISION POS` PALLET POSITION DOWN
      OUT     T4618 K3
      MPP
      AND     T4618
      AND     M21  ; AUTO MODE #2
      ANI     X52C  ; NG OUT UNIT DIVERTER PALLET DET
      AND     X52E  ; NG 배출 UNIT DIVERTER MID
      ANI     M4700  ; NG OUTLET CONV AUTO
      ANI     M4730  ; NG OUTLET.PALLET.PASS.AUTO
      OUT     T4623 K10
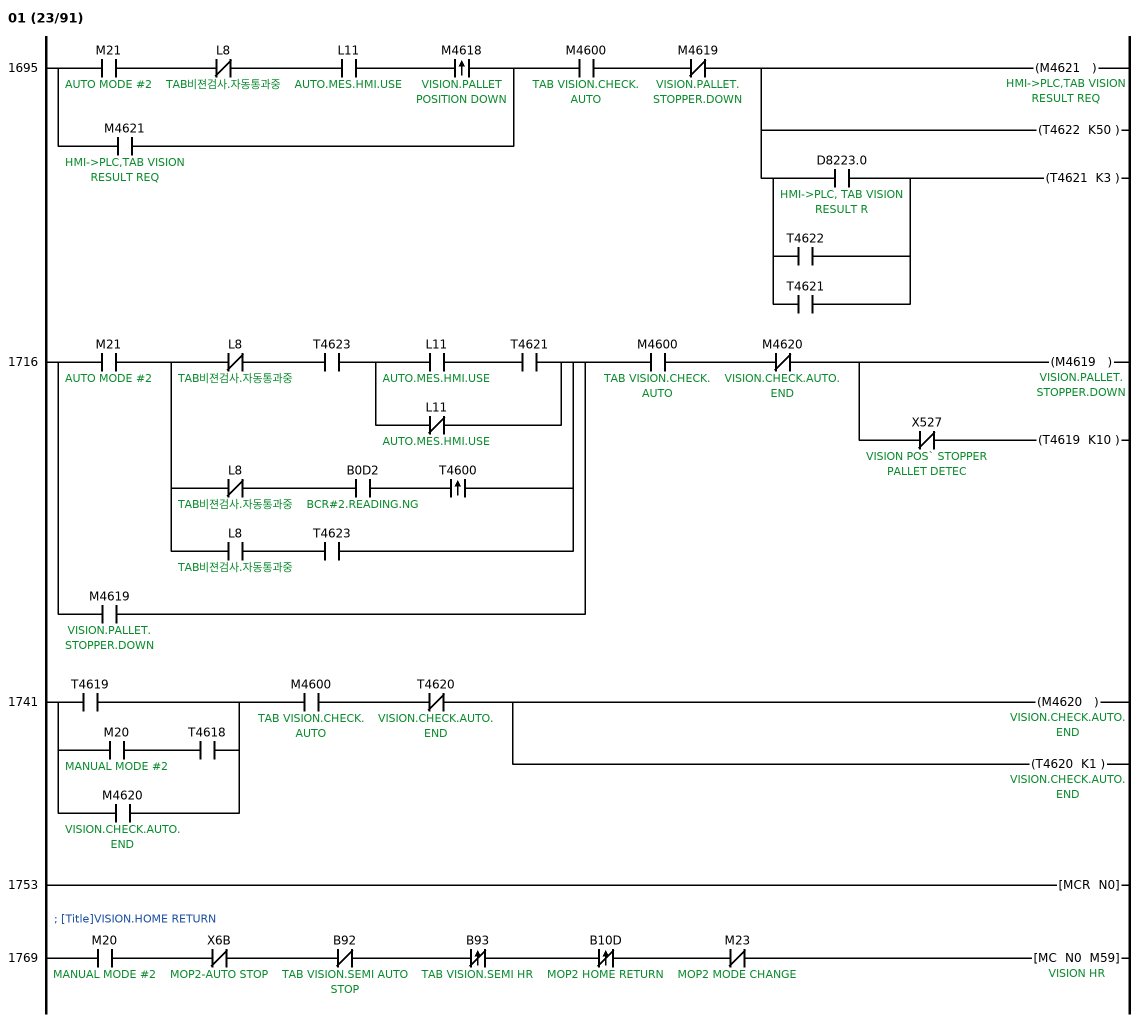
1695  LD      M21  ; AUTO MODE #2
      ANI     L8  ; TAB비젼검사.자동통과중
      AND     L11  ; AUTO.MES.HMI.USE
      ANDP    M4618  ; VISION.PALLET POSITION DOWN
      OR      M4621  ; HMI->PLC,TAB VISION RESULT REQ
      AND     M4600  ; TAB VISION.CHECK.AUTO
      ANI     M4619  ; VISION.PALLET.STOPPER.DOWN
      OUT     M4621  ; HMI->PLC,TAB VISION RESULT REQ
      OUT     T4622 K50
      LD      D8223.0  ; HMI->PLC, TAB VISION RESULT R
      OR      T4622
      OR      T4621
      ANB
      OUT     T4621 K3
1716  LD      M21  ; AUTO MODE #2
      LDI     L8  ; TAB비젼검사.자동통과중
      AND     T4623
      LD      L11  ; AUTO.MES.HMI.USE
      AND     T4621
      ORI     L11  ; AUTO.MES.HMI.USE
      ANB
      LDI     L8  ; TAB비젼검사.자동통과중
      AND     B0D2  ; BCR#2.READING.NG
      ANDP    T4600
      ORB
      LD      L8  ; TAB비젼검사.자동통과중
      AND     T4623
      ORB
      ANB
      OR      M4619  ; VISION.PALLET.STOPPER.DOWN
      AND     M4600  ; TAB VISION.CHECK.AUTO
      ANI     M4620  ; VISION.CHECK.AUTO.END
      OUT     M4619  ; VISION.PALLET.STOPPER.DOWN
      ANI     X527  ; VISION POS` STOPPER PALLET DETEC
      OUT     T4619 K10
1741  LD      T4619
      LD      M20  ; MANUAL MODE #2
      AND     T4618
      ORB
      OR      M4620  ; VISION.CHECK.AUTO.END
      AND     M4600  ; TAB VISION.CHECK.AUTO
      ANI     T4620  ; VISION.CHECK.AUTO.END
      OUT     M4620  ; VISION.CHECK.AUTO.END
      OUT     T4620 K1  ; VISION.CHECK.AUTO.END
1753  MCR     N0
; [Title]VISION.HOME RETURN
1769  LD      M20  ; MANUAL MODE #2
      ANI     X6B  ; MOP2-AUTO STOP
      ANI     B92  ; TAB VISION.SEMI AUTO STOP
      ANDPI   B93  ; TAB VISION.SEMI HR
      ANDPI   B10D  ; MOP2 HOME RETURN
      ANI     M23  ; MOP2 MODE CHANGE
      MC      N0 M59  ; VISION HR
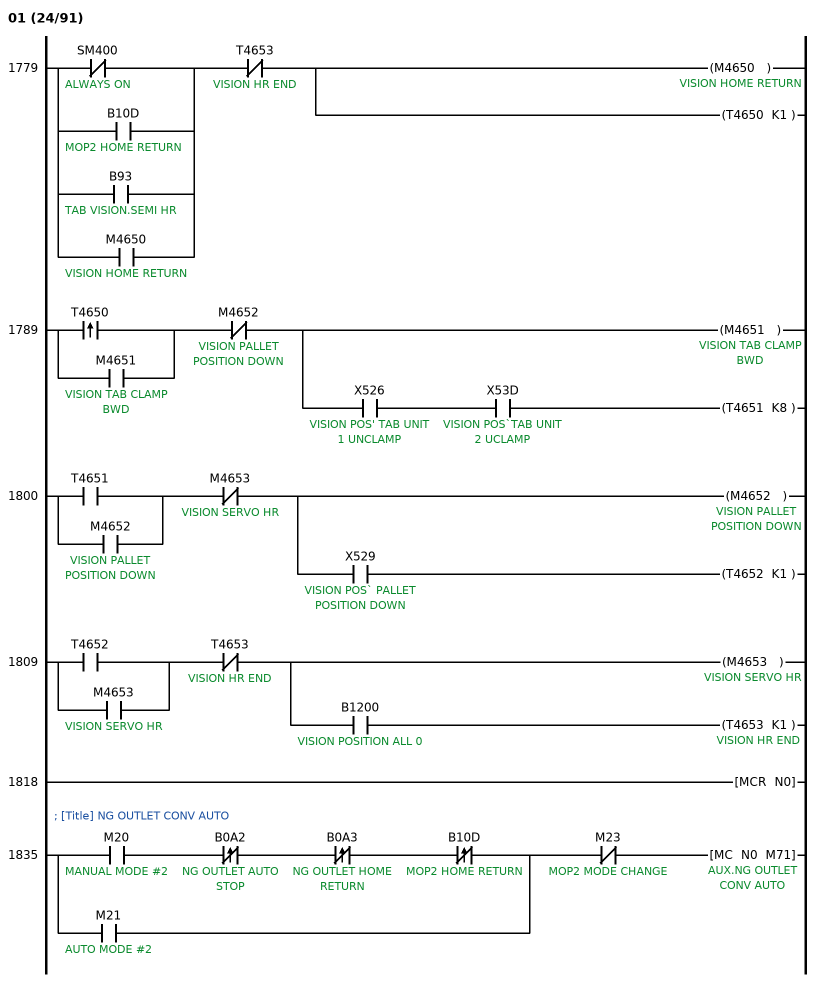
1779  LDI     SM400  ; ALWAYS ON
      OR      B10D  ; MOP2 HOME RETURN
      OR      B93  ; TAB VISION.SEMI HR
      OR      M4650  ; VISION HOME RETURN
      ANI     T4653  ; VISION HR END
      OUT     M4650  ; VISION HOME RETURN
      OUT     T4650 K1
1789  LDP     T4650
      OR      M4651  ; VISION TAB CLAMP BWD
      ANI     M4652  ; VISION PALLET POSITION DOWN
      OUT     M4651  ; VISION TAB CLAMP BWD
      AND     X526  ; VISION POS' TAB UNIT 1 UNCLAMP
      AND     X53D  ; VISION POS`TAB UNIT 2 UCLAMP
      OUT     T4651 K8
1800  LD      T4651
      OR      M4652  ; VISION PALLET POSITION DOWN
      ANI     M4653  ; VISION SERVO HR
      OUT     M4652  ; VISION PALLET POSITION DOWN
      AND     X529  ; VISION POS` PALLET POSITION DOWN
      OUT     T4652 K1
1809  LD      T4652
      OR      M4653  ; VISION SERVO HR
      ANI     T4653  ; VISION HR END
      OUT     M4653  ; VISION SERVO HR
      AND     B1200  ; VISION POSITION ALL 0
      OUT     T4653 K1  ; VISION HR END
1818  MCR     N0
; [Title] NG OUTLET CONV AUTO
1835  LD      M20  ; MANUAL MODE #2
      ANDPI   B0A2  ; NG OUTLET AUTO STOP
      ANDPI   B0A3  ; NG OUTLET HOME RETURN
      ANDPI   B10D  ; MOP2 HOME RETURN
      OR      M21  ; AUTO MODE #2
      ANI     M23  ; MOP2 MODE CHANGE
      MC      N0 M71  ; AUX.NG OUTLET CONV AUTO
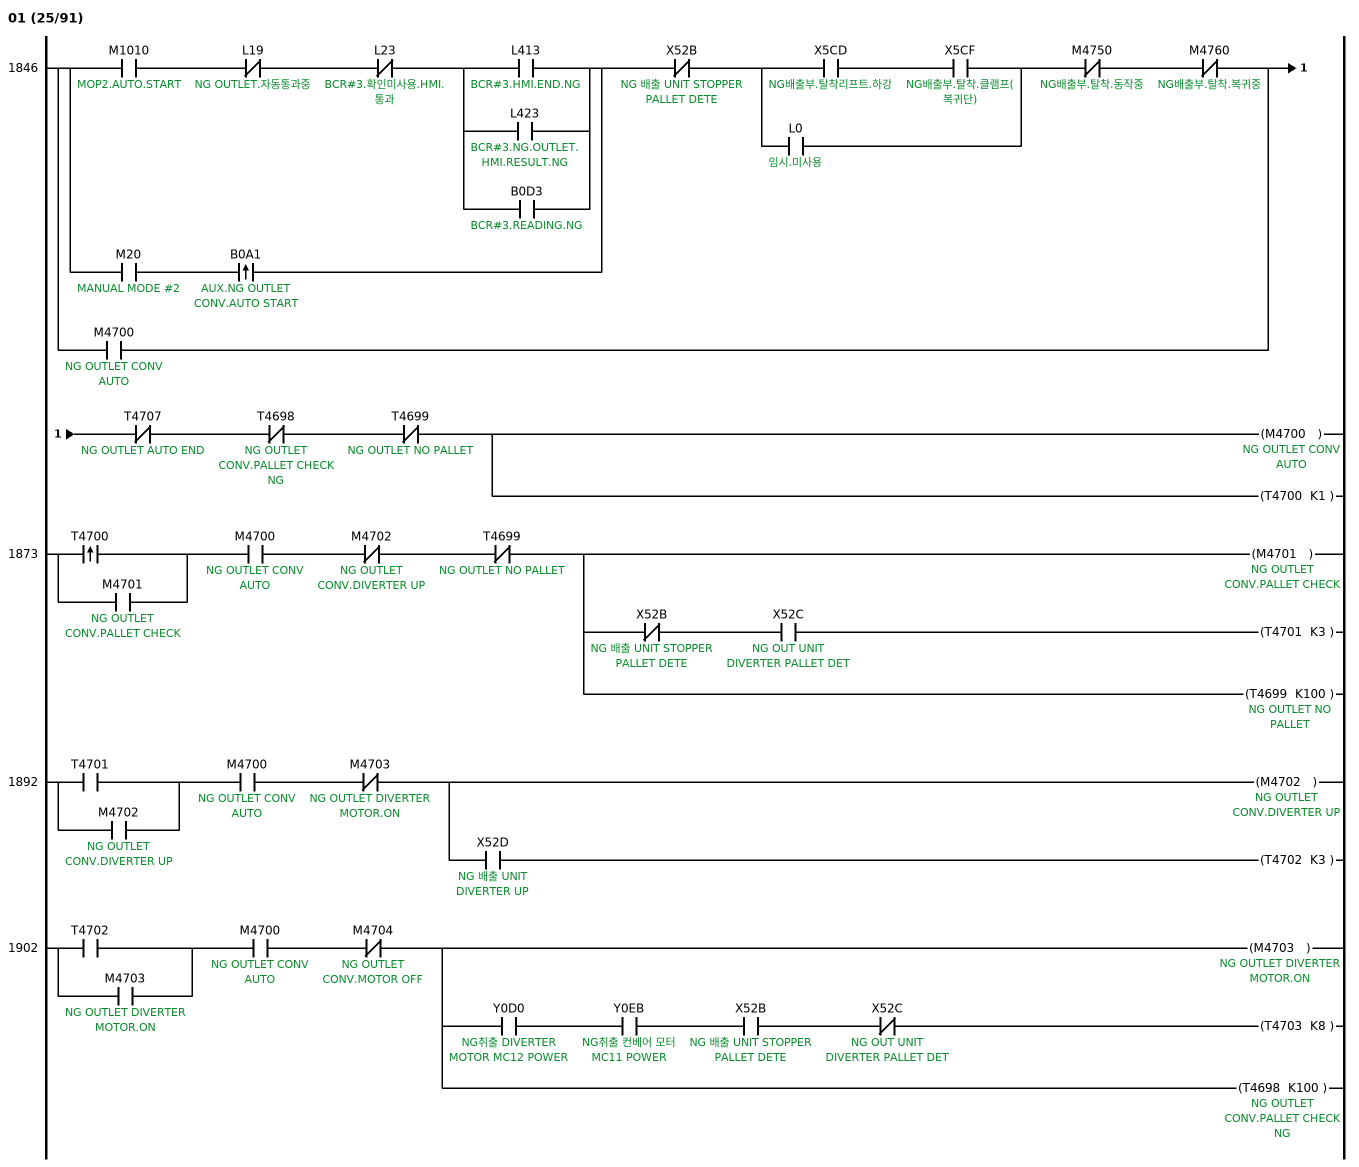
1846  LD      M1010  ; MOP2.AUTO.START
      ANI     L19  ; NG OUTLET.자동통과중
      ANI     L23  ; BCR#3.확인미사용.HMI.통과
      LD      L413  ; BCR#3.HMI.END.NG
      OR      L423  ; BCR#3.NG.OUTLET.HMI.RESULT.NG
      OR      B0D3  ; BCR#3.READING.NG
      ANB
      LD      M20  ; MANUAL MODE #2
      ANDP    B0A1  ; AUX.NG OUTLET CONV.AUTO START
      ORB
      ANI     X52B  ; NG 배출 UNIT STOPPER PALLET DETE
      LD      X5CD  ; NG배출부.탈착리프트.하강
      AND     X5CF  ; NG배출부.탈착.클램프(복귀단)
      OR      L0  ; 임시.미사용
      ANB
      ANI     M4750  ; NG배출부.탈착.동작중
      ANI     M4760  ; NG배출부.탈착.복귀중
      OR      M4700  ; NG OUTLET CONV AUTO
      ANI     T4707  ; NG OUTLET AUTO END
      ANI     T4698  ; NG OUTLET CONV.PALLET CHECK NG
      ANI     T4699  ; NG OUTLET NO PALLET
      OUT     M4700  ; NG OUTLET CONV AUTO
      OUT     T4700 K1
1873  LDP     T4700
      OR      M4701  ; NG OUTLET CONV.PALLET CHECK
      AND     M4700  ; NG OUTLET CONV AUTO
      ANI     M4702  ; NG OUTLET CONV.DIVERTER UP
      ANI     T4699  ; NG OUTLET NO PALLET
      OUT     M4701  ; NG OUTLET CONV.PALLET CHECK
      MPS
      ANI     X52B  ; NG 배출 UNIT STOPPER PALLET DETE
      AND     X52C  ; NG OUT UNIT DIVERTER PALLET DET
      OUT     T4701 K3
      MPP
      OUT     T4699 K100  ; NG OUTLET NO PALLET
1892  LD      T4701
      OR      M4702  ; NG OUTLET CONV.DIVERTER UP
      AND     M4700  ; NG OUTLET CONV AUTO
      ANI     M4703  ; NG OUTLET DIVERTER MOTOR.ON
      OUT     M4702  ; NG OUTLET CONV.DIVERTER UP
      AND     X52D  ; NG 배출 UNIT DIVERTER UP
      OUT     T4702 K3
1902  LD      T4702
      OR      M4703  ; NG OUTLET DIVERTER MOTOR.ON
      AND     M4700  ; NG OUTLET CONV AUTO
      ANI     M4704  ; NG OUTLET CONV.MOTOR OFF
      OUT     M4703  ; NG OUTLET DIVERTER MOTOR.ON
      MPS
      AND     Y0D0  ; NG취출 DIVERTER MOTOR MC12 POWER
      AND     Y0EB  ; NG취출 컨베어 모터 MC11 POWER
      AND     X52B  ; NG 배출 UNIT STOPPER PALLET DETE
      ANI     X52C  ; NG OUT UNIT DIVERTER PALLET DET
      OUT     T4703 K8
      MPP
      OUT     T4698 K100  ; NG OUTLET CONV.PALLET CHECK NG
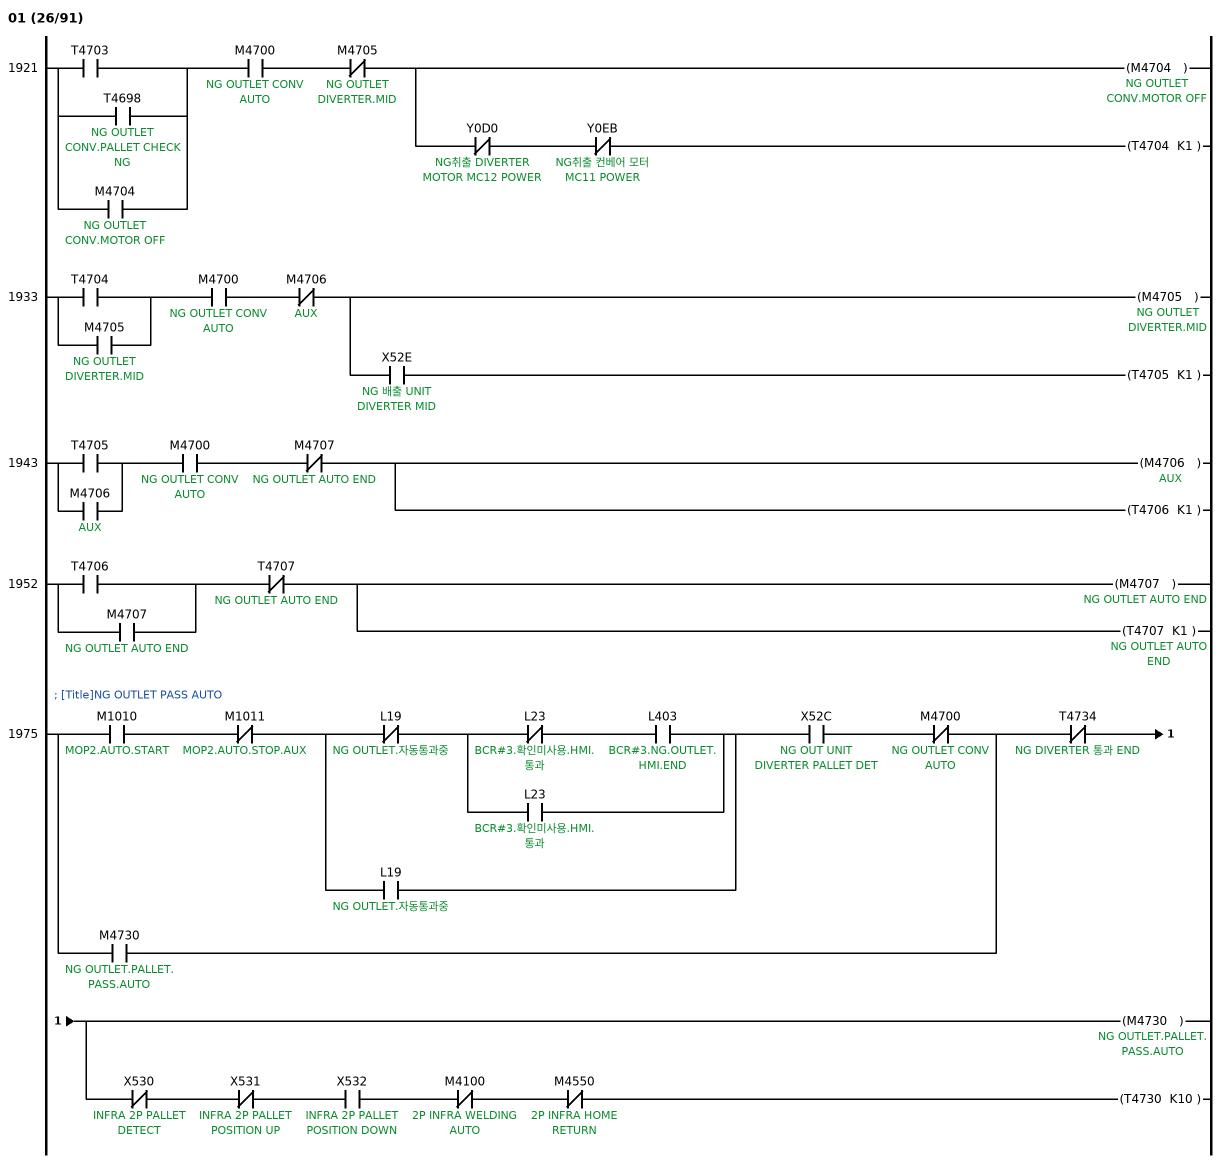
1921  LD      T4703
      OR      T4698  ; NG OUTLET CONV.PALLET CHECK NG
      OR      M4704  ; NG OUTLET CONV.MOTOR OFF
      AND     M4700  ; NG OUTLET CONV AUTO
      ANI     M4705  ; NG OUTLET DIVERTER.MID
      OUT     M4704  ; NG OUTLET CONV.MOTOR OFF
      ANI     Y0D0  ; NG취출 DIVERTER MOTOR MC12 POWER
      ANI     Y0EB  ; NG취출 컨베어 모터 MC11 POWER
      OUT     T4704 K1
1933  LD      T4704
      OR      M4705  ; NG OUTLET DIVERTER.MID
      AND     M4700  ; NG OUTLET CONV AUTO
      ANI     M4706  ; AUX
      OUT     M4705  ; NG OUTLET DIVERTER.MID
      AND     X52E  ; NG 배출 UNIT DIVERTER MID
      OUT     T4705 K1
1943  LD      T4705
      OR      M4706  ; AUX
      AND     M4700  ; NG OUTLET CONV AUTO
      ANI     M4707  ; NG OUTLET AUTO END
      OUT     M4706  ; AUX
      OUT     T4706 K1
1952  LD      T4706
      OR      M4707  ; NG OUTLET AUTO END
      ANI     T4707  ; NG OUTLET AUTO END
      OUT     M4707  ; NG OUTLET AUTO END
      OUT     T4707 K1  ; NG OUTLET AUTO END
; [Title]NG OUTLET PASS AUTO
1975  LD      M1010  ; MOP2.AUTO.START
      ANI     M1011  ; MOP2.AUTO.STOP.AUX
      LDI     L19  ; NG OUTLET.자동통과중
      LDI     L23  ; BCR#3.확인미사용.HMI.통과
      AND     L403  ; BCR#3.NG.OUTLET.HMI.END
      OR      L23  ; BCR#3.확인미사용.HMI.통과
      ANB
      OR      L19  ; NG OUTLET.자동통과중
      ANB
      AND     X52C  ; NG OUT UNIT DIVERTER PALLET DET
      ANI     M4700  ; NG OUTLET CONV AUTO
      OR      M4730  ; NG OUTLET.PALLET.PASS.AUTO
      ANI     T4734  ; NG DIVERTER 통과 END
      OUT     M4730  ; NG OUTLET.PALLET.PASS.AUTO
      ANI     X530  ; INFRA 2P PALLET DETECT
      ANI     X531  ; INFRA 2P PALLET POSITION UP
      AND     X532  ; INFRA 2P PALLET POSITION DOWN
      ANI     M4100  ; 2P INFRA WELDING AUTO
      ANI     M4550  ; 2P INFRA HOME RETURN
      OUT     T4730 K10
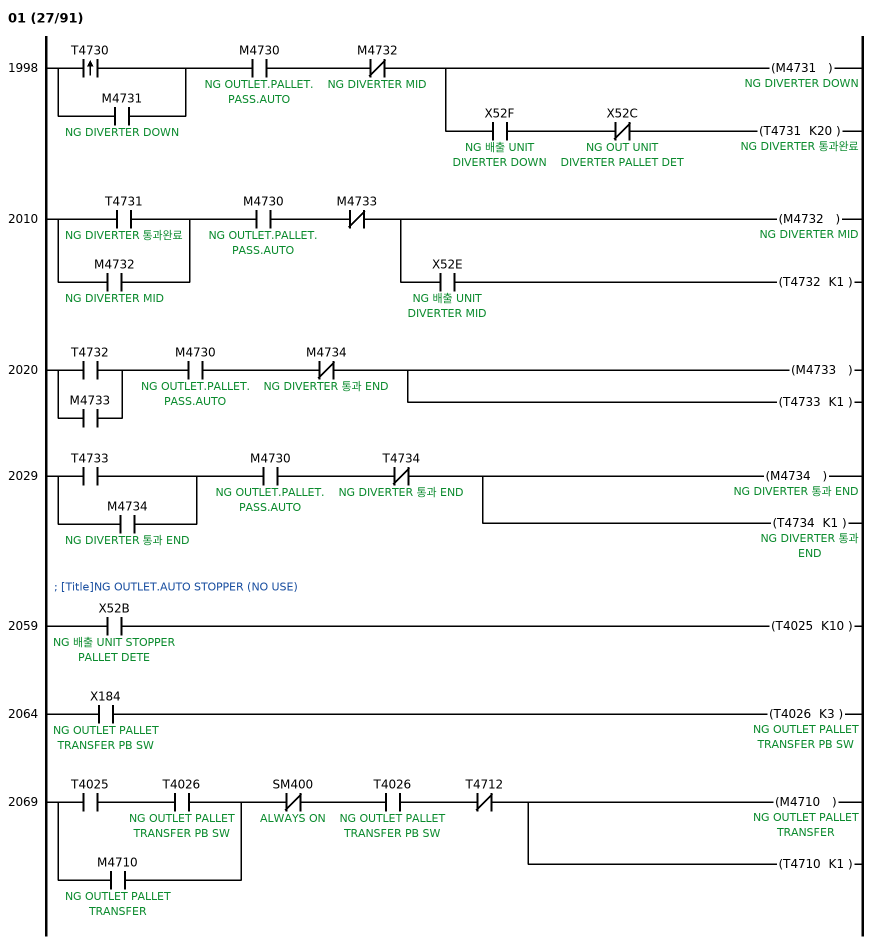
1998  LDP     T4730
      OR      M4731  ; NG DIVERTER DOWN
      AND     M4730  ; NG OUTLET.PALLET.PASS.AUTO
      ANI     M4732  ; NG DIVERTER MID
      OUT     M4731  ; NG DIVERTER DOWN
      AND     X52F  ; NG 배출 UNIT DIVERTER DOWN
      ANI     X52C  ; NG OUT UNIT DIVERTER PALLET DET
      OUT     T4731 K20  ; NG DIVERTER 통과완료
2010  LD      T4731  ; NG DIVERTER 통과완료
      OR      M4732  ; NG DIVERTER MID
      AND     M4730  ; NG OUTLET.PALLET.PASS.AUTO
      ANI     M4733
      OUT     M4732  ; NG DIVERTER MID
      AND     X52E  ; NG 배출 UNIT DIVERTER MID
      OUT     T4732 K1
2020  LD      T4732
      OR      M4733
      AND     M4730  ; NG OUTLET.PALLET.PASS.AUTO
      ANI     M4734  ; NG DIVERTER 통과 END
      OUT     M4733
      OUT     T4733 K1
2029  LD      T4733
      OR      M4734  ; NG DIVERTER 통과 END
      AND     M4730  ; NG OUTLET.PALLET.PASS.AUTO
      ANI     T4734  ; NG DIVERTER 통과 END
      OUT     M4734  ; NG DIVERTER 통과 END
      OUT     T4734 K1  ; NG DIVERTER 통과 END
; [Title]NG OUTLET.AUTO STOPPER (NO USE)
2059  LD      X52B  ; NG 배출 UNIT STOPPER PALLET DETE
      OUT     T4025 K10
2064  LD      X184  ; NG OUTLET PALLET TRANSFER PB SW
      OUT     T4026 K3  ; NG OUTLET PALLET TRANSFER PB SW
2069  LD      T4025
      AND     T4026  ; NG OUTLET PALLET TRANSFER PB SW
      OR      M4710  ; NG OUTLET PALLET TRANSFER
      ANI     SM400  ; ALWAYS ON
      AND     T4026  ; NG OUTLET PALLET TRANSFER PB SW
      ANI     T4712
      OUT     M4710  ; NG OUTLET PALLET TRANSFER
      OUT     T4710 K1
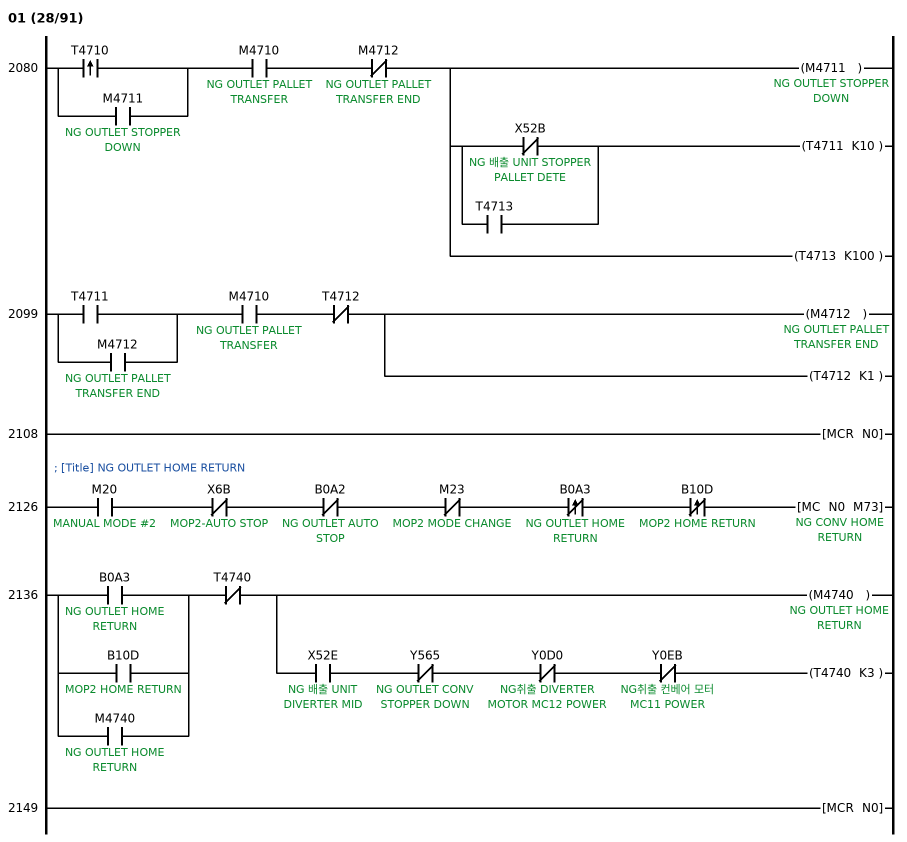
2080  LDP     T4710
      OR      M4711  ; NG OUTLET STOPPER DOWN
      AND     M4710  ; NG OUTLET PALLET TRANSFER
      ANI     M4712  ; NG OUTLET PALLET TRANSFER END
      OUT     M4711  ; NG OUTLET STOPPER DOWN
      MPS
      LDI     X52B  ; NG 배출 UNIT STOPPER PALLET DETE
      OR      T4713
      ANB
      OUT     T4711 K10
      MPP
      OUT     T4713 K100
2099  LD      T4711
      OR      M4712  ; NG OUTLET PALLET TRANSFER END
      AND     M4710  ; NG OUTLET PALLET TRANSFER
      ANI     T4712
      OUT     M4712  ; NG OUTLET PALLET TRANSFER END
      OUT     T4712 K1
2108  MCR     N0
; [Title] NG OUTLET HOME RETURN
2126  LD      M20  ; MANUAL MODE #2
      ANI     X6B  ; MOP2-AUTO STOP
      ANI     B0A2  ; NG OUTLET AUTO STOP
      ANI     M23  ; MOP2 MODE CHANGE
      ANDPI   B0A3  ; NG OUTLET HOME RETURN
      ANDPI   B10D  ; MOP2 HOME RETURN
      MC      N0 M73  ; NG CONV HOME RETURN
2136  LD      B0A3  ; NG OUTLET HOME RETURN
      OR      B10D  ; MOP2 HOME RETURN
      OR      M4740  ; NG OUTLET HOME RETURN
      ANI     T4740
      OUT     M4740  ; NG OUTLET HOME RETURN
      AND     X52E  ; NG 배출 UNIT DIVERTER MID
      ANI     Y565  ; NG OUTLET CONV STOPPER DOWN
      ANI     Y0D0  ; NG취출 DIVERTER MOTOR MC12 POWER
      ANI     Y0EB  ; NG취출 컨베어 모터 MC11 POWER
      OUT     T4740 K3
2149  MCR     N0
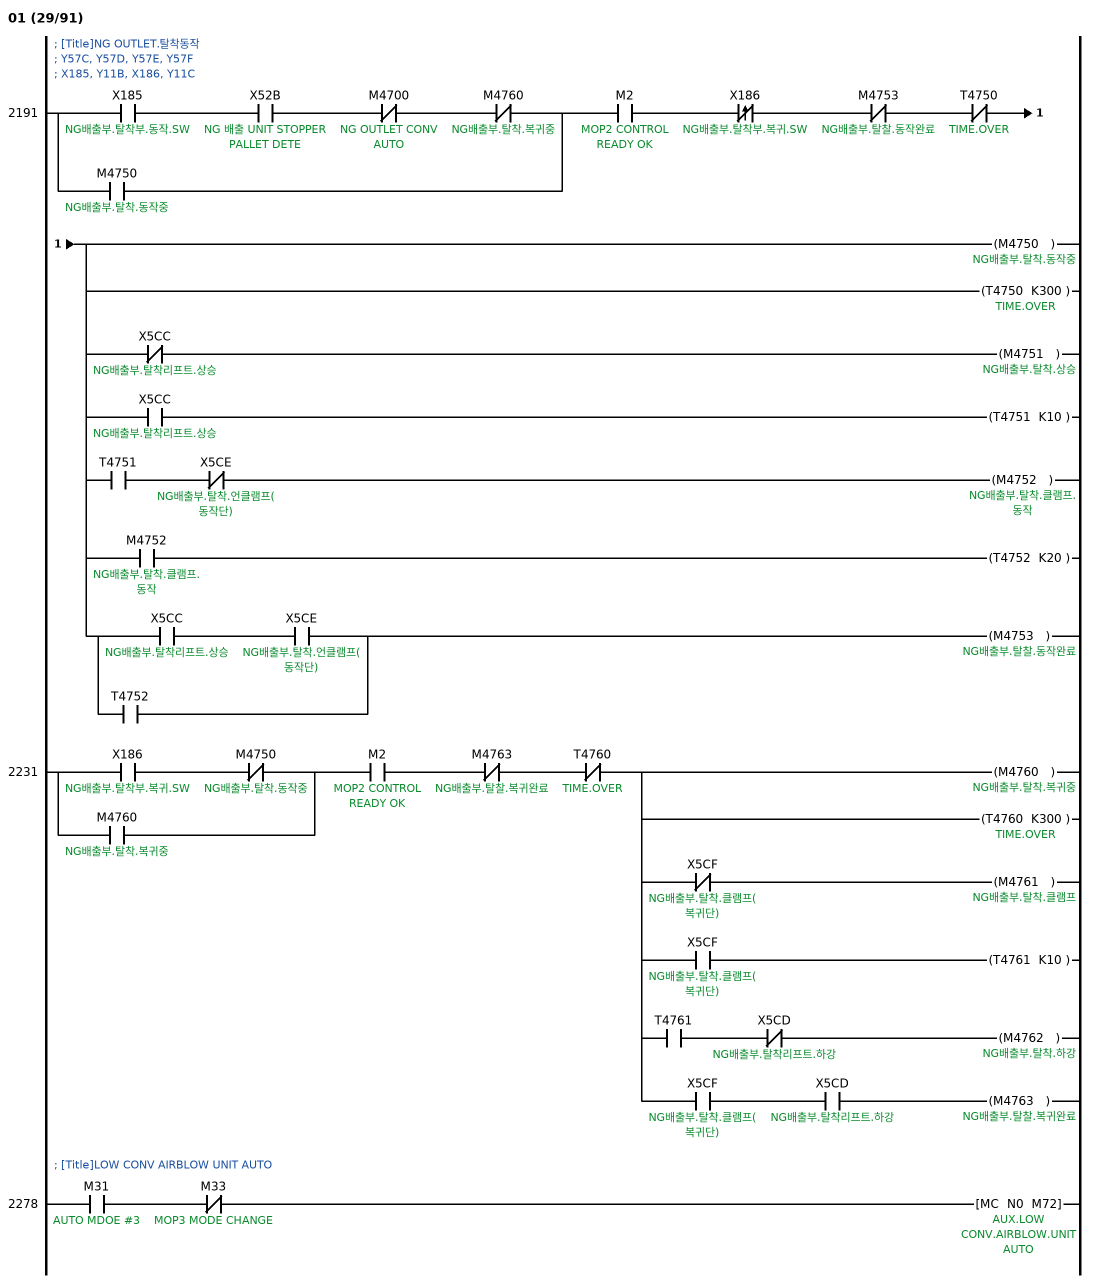
; [Title]NG OUTLET.탈착동작
; Y57C, Y57D, Y57E, Y57F
; X185, Y11B, X186, Y11C
2191  LD      X185  ; NG배출부.탈착부.동작.SW
      AND     X52B  ; NG 배출 UNIT STOPPER PALLET DETE
      ANI     M4700  ; NG OUTLET CONV AUTO
      ANI     M4760  ; NG배출부.탈착.복귀중
      OR      M4750  ; NG배출부.탈착.동작중
      AND     M2  ; MOP2 CONTROL READY OK
      ANDPI   X186  ; NG배출부.탈착부.복귀.SW
      ANI     M4753  ; NG배출부.탈찰.동작완료
      ANI     T4750  ; TIME.OVER
      OUT     M4750  ; NG배출부.탈착.동작중
      OUT     T4750 K300  ; TIME.OVER
      MPS
      ANI     X5CC  ; NG배출부.탈착리프트.상승
      OUT     M4751  ; NG배출부.탈착.상승
      MRD
      AND     X5CC  ; NG배출부.탈착리프트.상승
      OUT     T4751 K10
      MRD
      AND     T4751
      ANI     X5CE  ; NG배출부.탈착.언클램프(동작단)
      OUT     M4752  ; NG배출부.탈착.클램프.동작
      MRD
      AND     M4752  ; NG배출부.탈착.클램프.동작
      OUT     T4752 K20
      MPP
      LD      X5CC  ; NG배출부.탈착리프트.상승
      AND     X5CE  ; NG배출부.탈착.언클램프(동작단)
      OR      T4752
      ANB
      OUT     M4753  ; NG배출부.탈찰.동작완료
2231  LD      X186  ; NG배출부.탈착부.복귀.SW
      ANI     M4750  ; NG배출부.탈착.동작중
      OR      M4760  ; NG배출부.탈착.복귀중
      AND     M2  ; MOP2 CONTROL READY OK
      ANI     M4763  ; NG배출부.탈찰.복귀완료
      ANI     T4760  ; TIME.OVER
      OUT     M4760  ; NG배출부.탈착.복귀중
      OUT     T4760 K300  ; TIME.OVER
      MPS
      ANI     X5CF  ; NG배출부.탈착.클램프(복귀단)
      OUT     M4761  ; NG배출부.탈착.클램프
      MRD
      AND     X5CF  ; NG배출부.탈착.클램프(복귀단)
      OUT     T4761 K10
      MRD
      AND     T4761
      ANI     X5CD  ; NG배출부.탈착리프트.하강
      OUT     M4762  ; NG배출부.탈착.하강
      MPP
      AND     X5CF  ; NG배출부.탈착.클램프(복귀단)
      AND     X5CD  ; NG배출부.탈착리프트.하강
      OUT     M4763  ; NG배출부.탈찰.복귀완료
; [Title]LOW CONV AIRBLOW UNIT AUTO
2278  LD      M31  ; AUTO MDOE #3
      ANI     M33  ; MOP3 MODE CHANGE
      MC      N0 M72  ; AUX.LOW CONV.AIRBLOW.UNIT AUTO
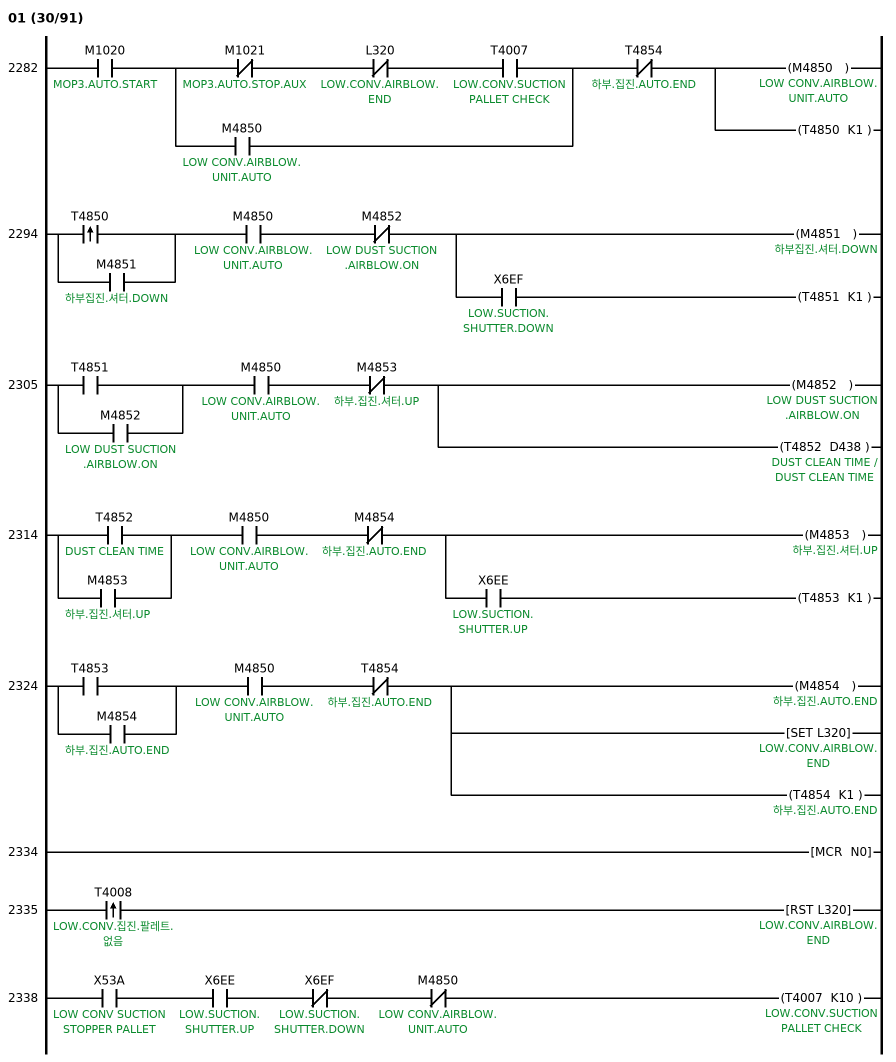
2282  LD      M1020  ; MOP3.AUTO.START
      LDI     M1021  ; MOP3.AUTO.STOP.AUX
      ANI     L320  ; LOW.CONV.AIRBLOW.END
      AND     T4007  ; LOW.CONV.SUCTION PALLET CHECK
      OR      M4850  ; LOW CONV.AIRBLOW.UNIT.AUTO
      ANB
      ANI     T4854  ; 하부.집진.AUTO.END
      OUT     M4850  ; LOW CONV.AIRBLOW.UNIT.AUTO
      OUT     T4850 K1
2294  LDP     T4850
      OR      M4851  ; 하부집진.셔터.DOWN
      AND     M4850  ; LOW CONV.AIRBLOW.UNIT.AUTO
      ANI     M4852  ; LOW DUST SUCTION .AIRBLOW.ON
      OUT     M4851  ; 하부집진.셔터.DOWN
      AND     X6EF  ; LOW.SUCTION.SHUTTER.DOWN
      OUT     T4851 K1
2305  LD      T4851
      OR      M4852  ; LOW DUST SUCTION .AIRBLOW.ON
      AND     M4850  ; LOW CONV.AIRBLOW.UNIT.AUTO
      ANI     M4853  ; 하부.집진.셔터.UP
      OUT     M4852  ; LOW DUST SUCTION .AIRBLOW.ON
      OUT     T4852 D438  ; DUST CLEAN TIME / DUST CLEAN TIME
2314  LD      T4852  ; DUST CLEAN TIME
      OR      M4853  ; 하부.집진.셔터.UP
      AND     M4850  ; LOW CONV.AIRBLOW.UNIT.AUTO
      ANI     M4854  ; 하부.집진.AUTO.END
      OUT     M4853  ; 하부.집진.셔터.UP
      AND     X6EE  ; LOW.SUCTION.SHUTTER.UP
      OUT     T4853 K1
2324  LD      T4853
      OR      M4854  ; 하부.집진.AUTO.END
      AND     M4850  ; LOW CONV.AIRBLOW.UNIT.AUTO
      ANI     T4854  ; 하부.집진.AUTO.END
      OUT     M4854  ; 하부.집진.AUTO.END
      SET     L320  ; LOW.CONV.AIRBLOW.END
      OUT     T4854 K1  ; 하부.집진.AUTO.END
2334  MCR     N0
2335  LDP     T4008  ; LOW.CONV.집진.팔레트.없음
      RST     L320  ; LOW.CONV.AIRBLOW.END
2338  LD      X53A  ; LOW CONV SUCTION STOPPER PALLET
      AND     X6EE  ; LOW.SUCTION.SHUTTER.UP
      ANI     X6EF  ; LOW.SUCTION.SHUTTER.DOWN
      ANI     M4850  ; LOW CONV.AIRBLOW.UNIT.AUTO
      OUT     T4007 K10  ; LOW.CONV.SUCTION PALLET CHECK
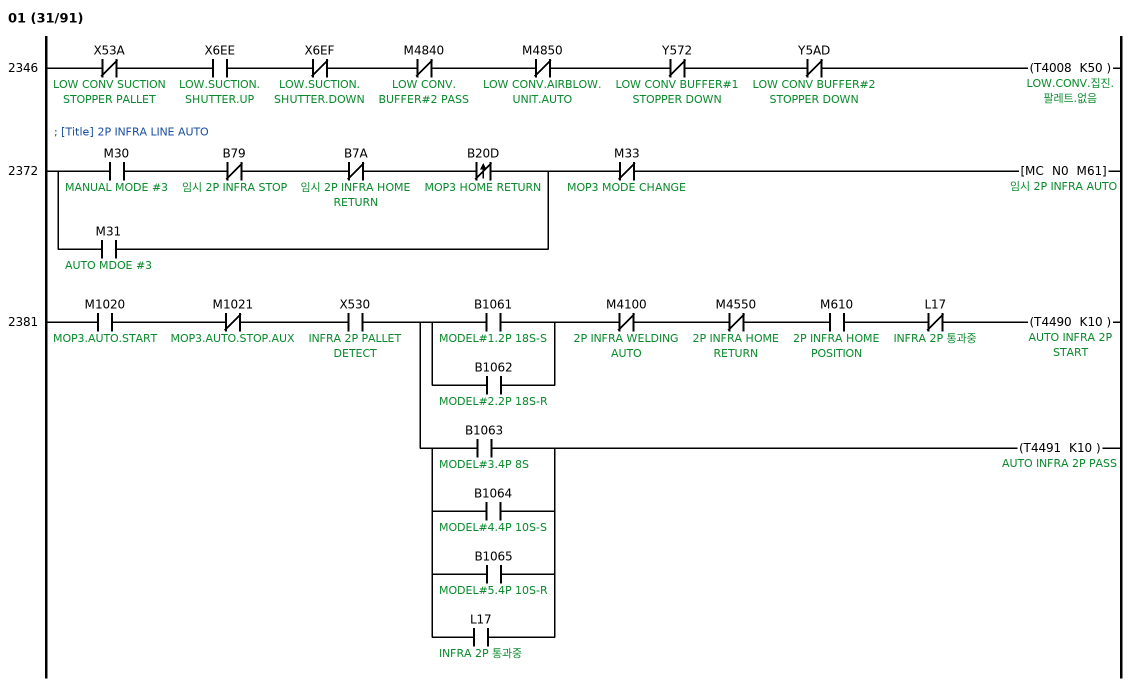
2346  LDI     X53A  ; LOW CONV SUCTION STOPPER PALLET
      AND     X6EE  ; LOW.SUCTION.SHUTTER.UP
      ANI     X6EF  ; LOW.SUCTION.SHUTTER.DOWN
      ANI     M4840  ; LOW CONV. BUFFER#2 PASS
      ANI     M4850  ; LOW CONV.AIRBLOW.UNIT.AUTO
      ANI     Y572  ; LOW CONV BUFFER#1 STOPPER DOWN
      ANI     Y5AD  ; LOW CONV BUFFER#2 STOPPER DOWN
      OUT     T4008 K50  ; LOW.CONV.집진.팔레트.없음
; [Title] 2P INFRA LINE AUTO
2372  LD      M30  ; MANUAL MODE #3
      ANI     B79  ; 임시 2P INFRA STOP
      ANI     B7A  ; 임시 2P INFRA HOME RETURN
      ANDPI   B20D  ; MOP3 HOME RETURN
      OR      M31  ; AUTO MDOE #3
      ANI     M33  ; MOP3 MODE CHANGE
      MC      N0 M61  ; 임시 2P INFRA AUTO
2381  LD      M1020  ; MOP3.AUTO.START
      ANI     M1021  ; MOP3.AUTO.STOP.AUX
      AND     X530  ; INFRA 2P PALLET DETECT
      MPS
      LD      B1061  ; MODEL#1.2P 18S-S
      OR      B1062  ; MODEL#2.2P 18S-R
      ANB
      ANI     M4100  ; 2P INFRA WELDING AUTO
      ANI     M4550  ; 2P INFRA HOME RETURN
      AND     M610  ; 2P INFRA HOME POSITION
      ANI     L17  ; INFRA 2P 통과중
      OUT     T4490 K10  ; AUTO INFRA 2P START
      MPP
      LD      B1063  ; MODEL#3.4P 8S
      OR      B1064  ; MODEL#4.4P 10S-S
      OR      B1065  ; MODEL#5.4P 10S-R
      OR      L17  ; INFRA 2P 통과중
      ANB
      OUT     T4491 K10  ; AUTO INFRA 2P PASS
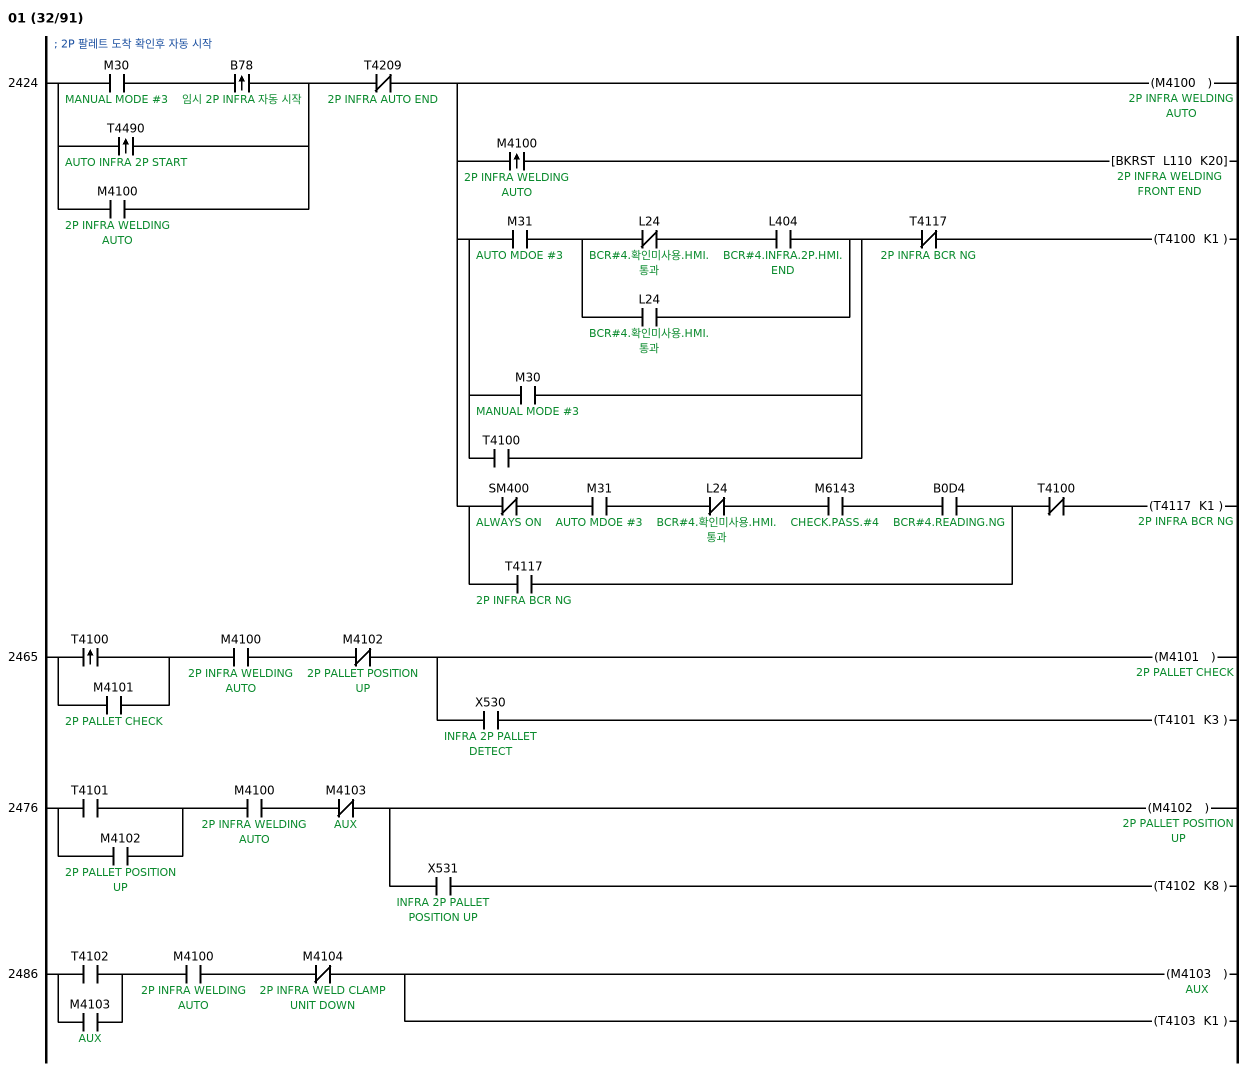
; 2P 팔레트 도착 확인후 자동 시작
2424  LD      M30  ; MANUAL MODE #3
      ANDP    B78  ; 임시 2P INFRA 자동 시작
      ORP     T4490  ; AUTO INFRA 2P START
      OR      M4100  ; 2P INFRA WELDING AUTO
      ANI     T4209  ; 2P INFRA AUTO END
      OUT     M4100  ; 2P INFRA WELDING AUTO
      MPS
      ANDP    M4100  ; 2P INFRA WELDING AUTO
      BKRST   L110 K20  ; 2P INFRA WELDING FRONT END
      MRD
      LD      M31  ; AUTO MDOE #3
      LDI     L24  ; BCR#4.확인미사용.HMI.통과
      AND     L404  ; BCR#4.INFRA.2P.HMI.END
      OR      L24  ; BCR#4.확인미사용.HMI.통과
      ANB
      OR      M30  ; MANUAL MODE #3
      OR      T4100
      ANB
      ANI     T4117  ; 2P INFRA BCR NG
      OUT     T4100 K1
      MPP
      LDI     SM400  ; ALWAYS ON
      AND     M31  ; AUTO MDOE #3
      ANI     L24  ; BCR#4.확인미사용.HMI.통과
      AND     M6143  ; CHECK.PASS.#4
      AND     B0D4  ; BCR#4.READING.NG
      OR      T4117  ; 2P INFRA BCR NG
      ANB
      ANI     T4100
      OUT     T4117 K1  ; 2P INFRA BCR NG
2465  LDP     T4100
      OR      M4101  ; 2P PALLET CHECK
      AND     M4100  ; 2P INFRA WELDING AUTO
      ANI     M4102  ; 2P PALLET POSITION UP
      OUT     M4101  ; 2P PALLET CHECK
      AND     X530  ; INFRA 2P PALLET DETECT
      OUT     T4101 K3
2476  LD      T4101
      OR      M4102  ; 2P PALLET POSITION UP
      AND     M4100  ; 2P INFRA WELDING AUTO
      ANI     M4103  ; AUX
      OUT     M4102  ; 2P PALLET POSITION UP
      AND     X531  ; INFRA 2P PALLET POSITION UP
      OUT     T4102 K8
2486  LD      T4102
      OR      M4103  ; AUX
      AND     M4100  ; 2P INFRA WELDING AUTO
      ANI     M4104  ; 2P INFRA WELD CLAMP UNIT DOWN
      OUT     M4103  ; AUX
      OUT     T4103 K1
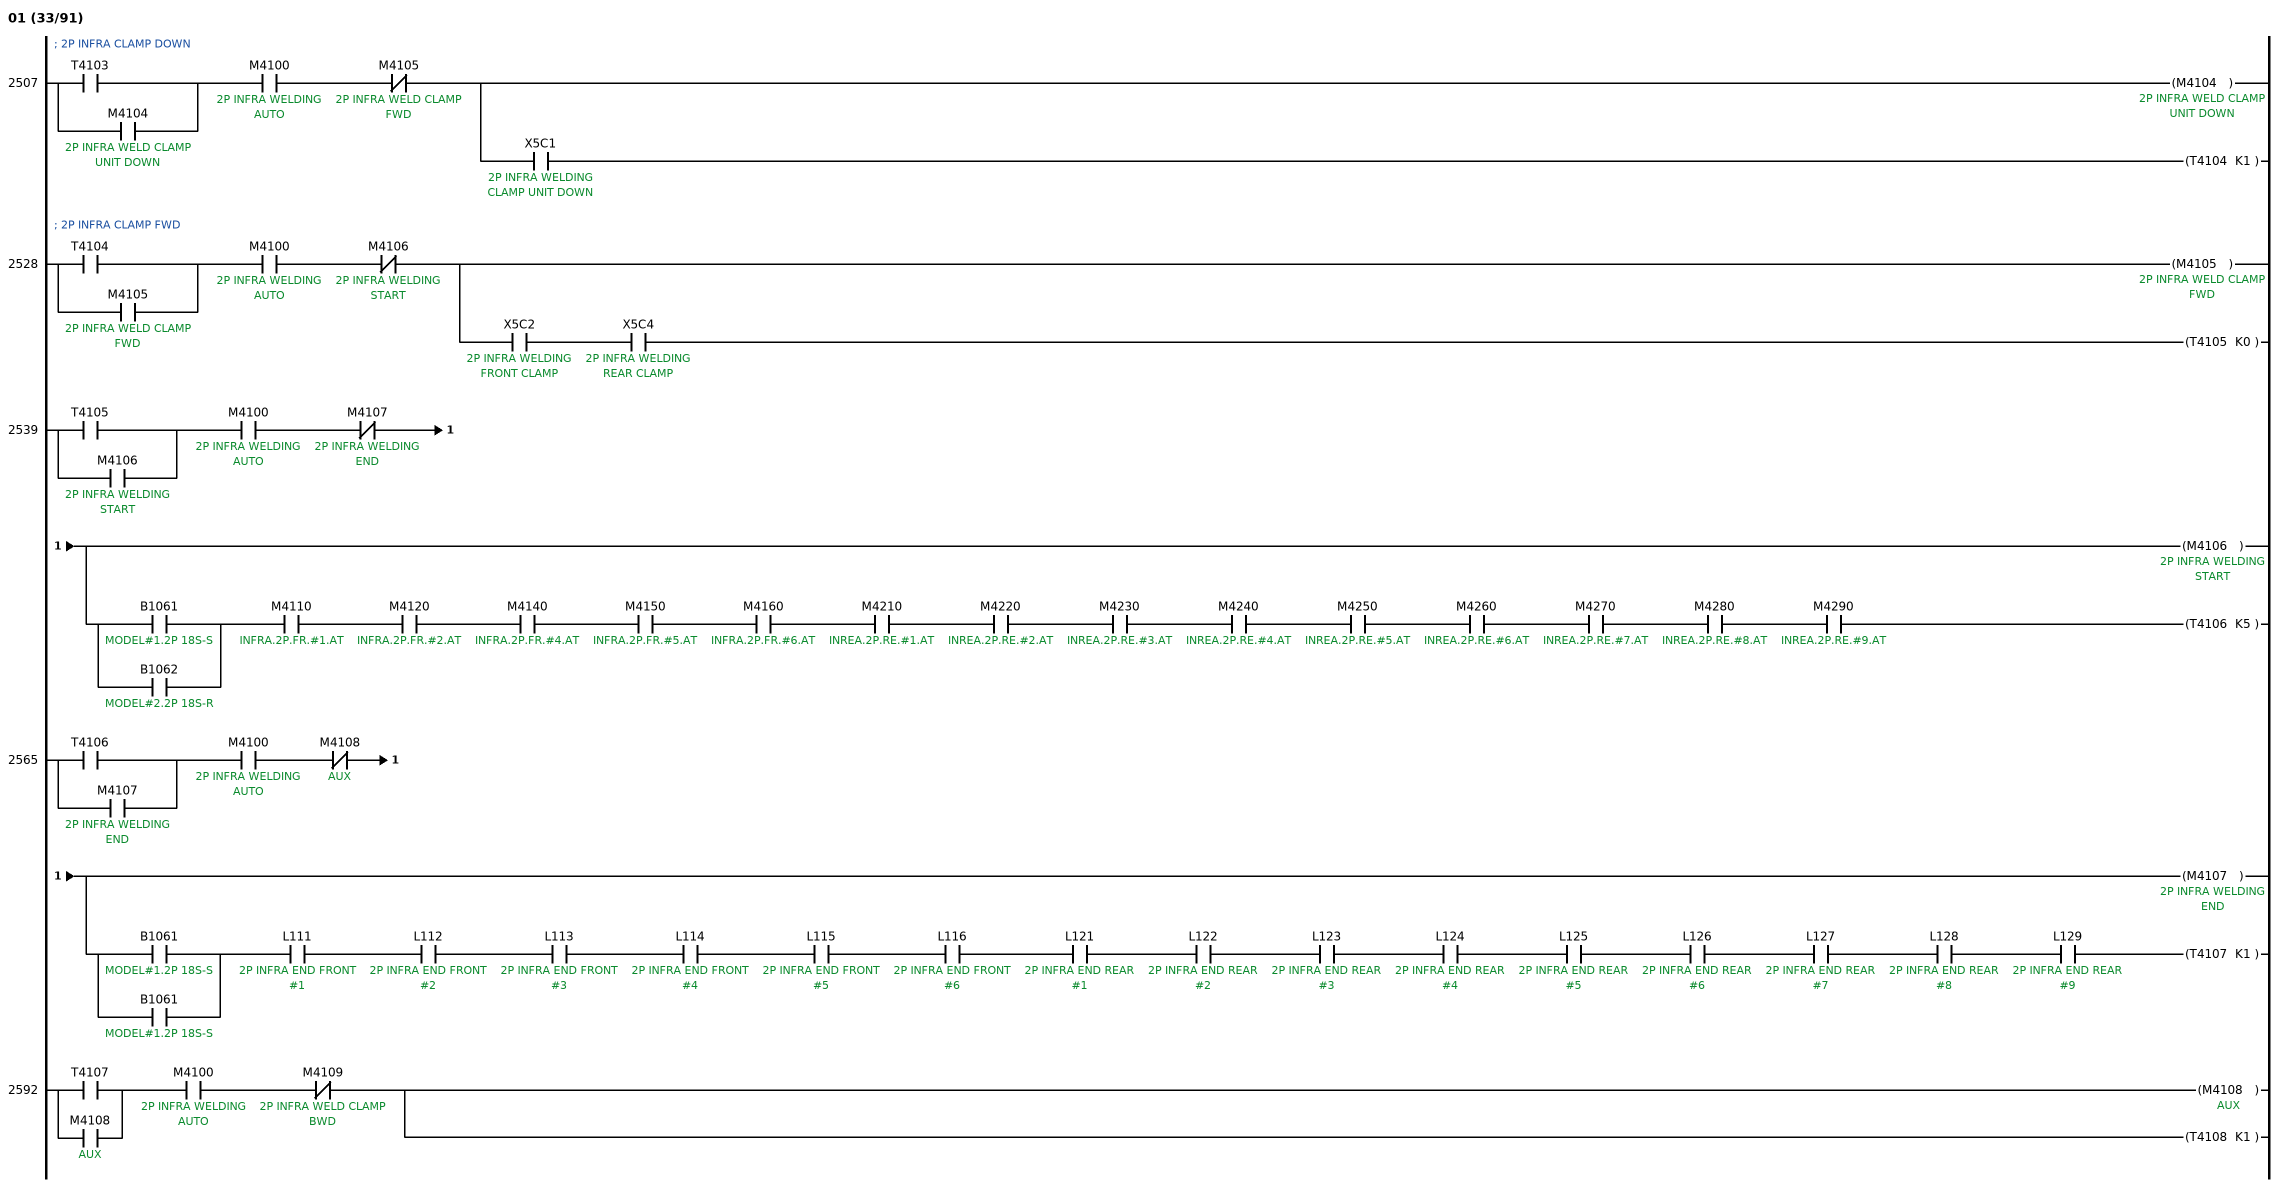
; 2P INFRA CLAMP DOWN
2507  LD      T4103
      OR      M4104  ; 2P INFRA WELD CLAMP UNIT DOWN
      AND     M4100  ; 2P INFRA WELDING AUTO
      ANI     M4105  ; 2P INFRA WELD CLAMP FWD
      OUT     M4104  ; 2P INFRA WELD CLAMP UNIT DOWN
      AND     X5C1  ; 2P INFRA WELDING CLAMP UNIT DOWN
      OUT     T4104 K1
; 2P INFRA CLAMP FWD
2528  LD      T4104
      OR      M4105  ; 2P INFRA WELD CLAMP FWD
      AND     M4100  ; 2P INFRA WELDING AUTO
      ANI     M4106  ; 2P INFRA WELDING START
      OUT     M4105  ; 2P INFRA WELD CLAMP FWD
      AND     X5C2  ; 2P INFRA WELDING FRONT CLAMP
      AND     X5C4  ; 2P INFRA WELDING REAR CLAMP
      OUT     T4105 K0
2539  LD      T4105
      OR      M4106  ; 2P INFRA WELDING START
      AND     M4100  ; 2P INFRA WELDING AUTO
      ANI     M4107  ; 2P INFRA WELDING END
      OUT     M4106  ; 2P INFRA WELDING START
      LD      B1061  ; MODEL#1.2P 18S-S
      OR      B1062  ; MODEL#2.2P 18S-R
      ANB
      AND     M4110  ; INFRA.2P.FR.#1.AT
      AND     M4120  ; INFRA.2P.FR.#2.AT
      AND     M4140  ; INFRA.2P.FR.#4.AT
      AND     M4150  ; INFRA.2P.FR.#5.AT
      AND     M4160  ; INFRA.2P.FR.#6.AT
      AND     M4210  ; INREA.2P.RE.#1.AT
      AND     M4220  ; INREA.2P.RE.#2.AT
      AND     M4230  ; INREA.2P.RE.#3.AT
      AND     M4240  ; INREA.2P.RE.#4.AT
      AND     M4250  ; INREA.2P.RE.#5.AT
      AND     M4260  ; INREA.2P.RE.#6.AT
      AND     M4270  ; INREA.2P.RE.#7.AT
      AND     M4280  ; INREA.2P.RE.#8.AT
      AND     M4290  ; INREA.2P.RE.#9.AT
      OUT     T4106 K5
2565  LD      T4106
      OR      M4107  ; 2P INFRA WELDING END
      AND     M4100  ; 2P INFRA WELDING AUTO
      ANI     M4108  ; AUX
      OUT     M4107  ; 2P INFRA WELDING END
      LD      B1061  ; MODEL#1.2P 18S-S
      OR      B1061  ; MODEL#1.2P 18S-S
      ANB
      AND     L111  ; 2P INFRA END FRONT #1
      AND     L112  ; 2P INFRA END FRONT #2
      AND     L113  ; 2P INFRA END FRONT #3
      AND     L114  ; 2P INFRA END FRONT #4
      AND     L115  ; 2P INFRA END FRONT #5
      AND     L116  ; 2P INFRA END FRONT #6
      AND     L121  ; 2P INFRA END REAR #1
      AND     L122  ; 2P INFRA END REAR #2
      AND     L123  ; 2P INFRA END REAR #3
      AND     L124  ; 2P INFRA END REAR #4
      AND     L125  ; 2P INFRA END REAR #5
      AND     L126  ; 2P INFRA END REAR #6
      AND     L127  ; 2P INFRA END REAR #7
      AND     L128  ; 2P INFRA END REAR #8
      AND     L129  ; 2P INFRA END REAR #9
      OUT     T4107 K1
2592  LD      T4107
      OR      M4108  ; AUX
      AND     M4100  ; 2P INFRA WELDING AUTO
      ANI     M4109  ; 2P INFRA WELD CLAMP BWD
      OUT     M4108  ; AUX
      OUT     T4108 K1
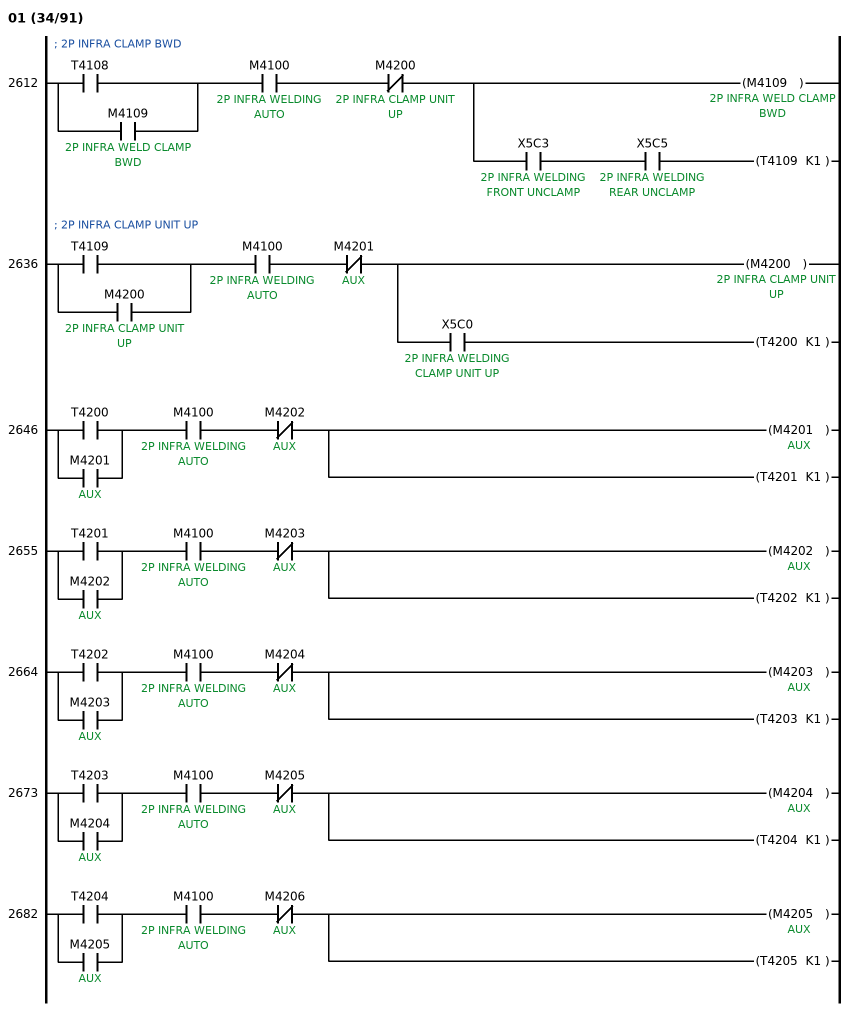
; 2P INFRA CLAMP BWD
2612  LD      T4108
      OR      M4109  ; 2P INFRA WELD CLAMP BWD
      AND     M4100  ; 2P INFRA WELDING AUTO
      ANI     M4200  ; 2P INFRA CLAMP UNIT UP
      OUT     M4109  ; 2P INFRA WELD CLAMP BWD
      AND     X5C3  ; 2P INFRA WELDING FRONT UNCLAMP
      AND     X5C5  ; 2P INFRA WELDING REAR UNCLAMP
      OUT     T4109 K1
; 2P INFRA CLAMP UNIT UP
2636  LD      T4109
      OR      M4200  ; 2P INFRA CLAMP UNIT UP
      AND     M4100  ; 2P INFRA WELDING AUTO
      ANI     M4201  ; AUX
      OUT     M4200  ; 2P INFRA CLAMP UNIT UP
      AND     X5C0  ; 2P INFRA WELDING CLAMP UNIT UP
      OUT     T4200 K1
2646  LD      T4200
      OR      M4201  ; AUX
      AND     M4100  ; 2P INFRA WELDING AUTO
      ANI     M4202  ; AUX
      OUT     M4201  ; AUX
      OUT     T4201 K1
2655  LD      T4201
      OR      M4202  ; AUX
      AND     M4100  ; 2P INFRA WELDING AUTO
      ANI     M4203  ; AUX
      OUT     M4202  ; AUX
      OUT     T4202 K1
2664  LD      T4202
      OR      M4203  ; AUX
      AND     M4100  ; 2P INFRA WELDING AUTO
      ANI     M4204  ; AUX
      OUT     M4203  ; AUX
      OUT     T4203 K1
2673  LD      T4203
      OR      M4204  ; AUX
      AND     M4100  ; 2P INFRA WELDING AUTO
      ANI     M4205  ; AUX
      OUT     M4204  ; AUX
      OUT     T4204 K1
2682  LD      T4204
      OR      M4205  ; AUX
      AND     M4100  ; 2P INFRA WELDING AUTO
      ANI     M4206  ; AUX
      OUT     M4205  ; AUX
      OUT     T4205 K1
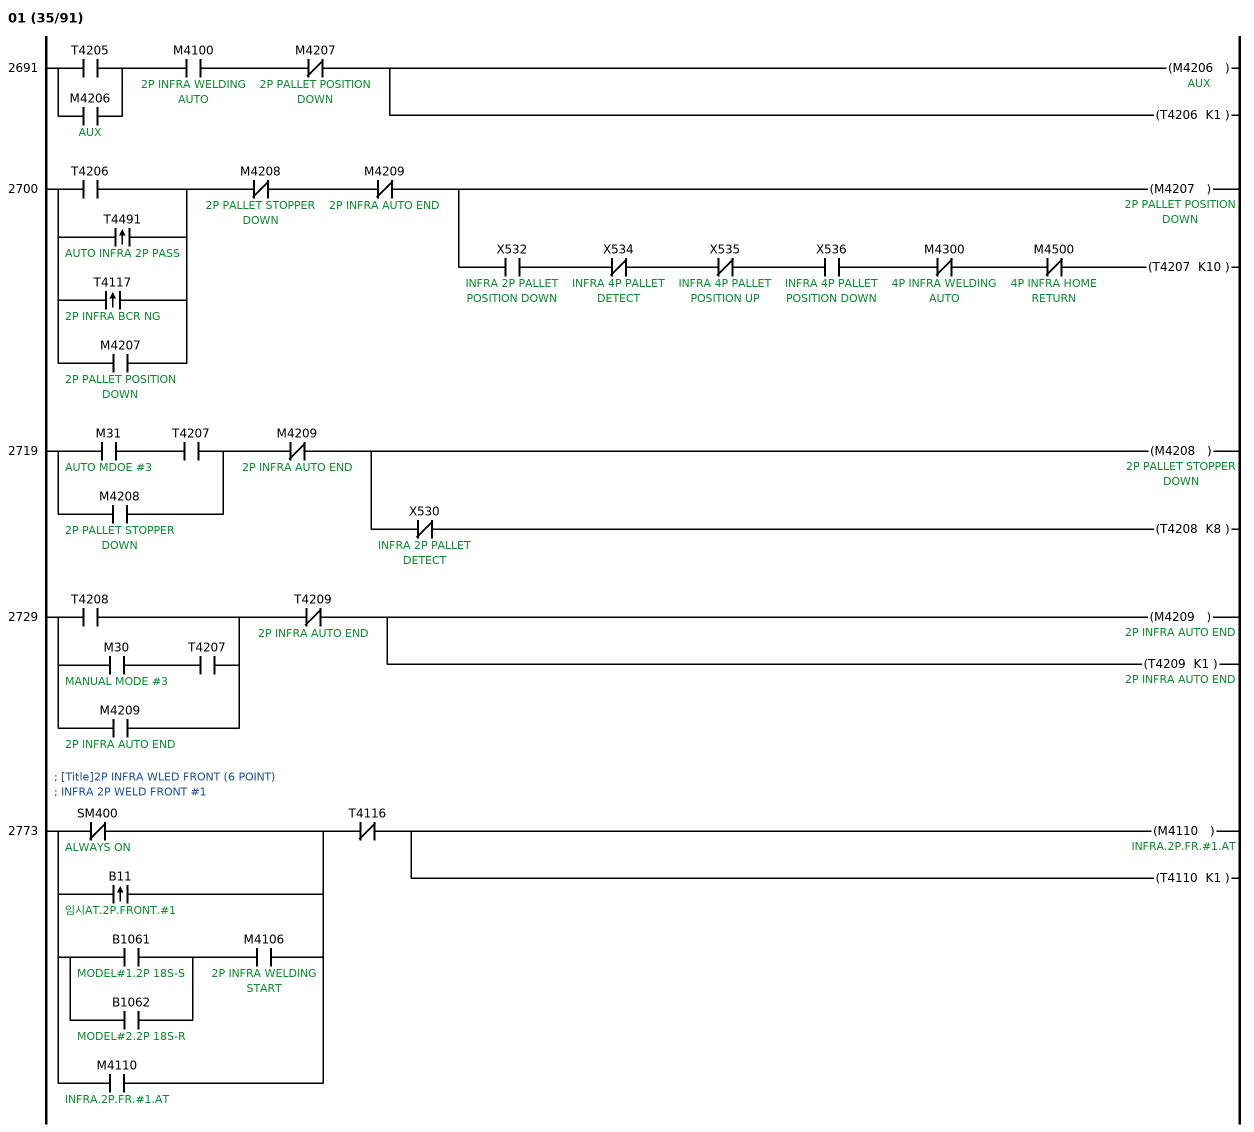
2691  LD      T4205
      OR      M4206  ; AUX
      AND     M4100  ; 2P INFRA WELDING AUTO
      ANI     M4207  ; 2P PALLET POSITION DOWN
      OUT     M4206  ; AUX
      OUT     T4206 K1
2700  LD      T4206
      ORP     T4491  ; AUTO INFRA 2P PASS
      ORP     T4117  ; 2P INFRA BCR NG
      OR      M4207  ; 2P PALLET POSITION DOWN
      ANI     M4208  ; 2P PALLET STOPPER DOWN
      ANI     M4209  ; 2P INFRA AUTO END
      OUT     M4207  ; 2P PALLET POSITION DOWN
      AND     X532  ; INFRA 2P PALLET POSITION DOWN
      ANI     X534  ; INFRA 4P PALLET DETECT
      ANI     X535  ; INFRA 4P PALLET POSITION UP
      AND     X536  ; INFRA 4P PALLET POSITION DOWN
      ANI     M4300  ; 4P INFRA WELDING AUTO
      ANI     M4500  ; 4P INFRA HOME RETURN
      OUT     T4207 K10
2719  LD      M31  ; AUTO MDOE #3
      AND     T4207
      OR      M4208  ; 2P PALLET STOPPER DOWN
      ANI     M4209  ; 2P INFRA AUTO END
      OUT     M4208  ; 2P PALLET STOPPER DOWN
      ANI     X530  ; INFRA 2P PALLET DETECT
      OUT     T4208 K8
2729  LD      T4208
      LD      M30  ; MANUAL MODE #3
      AND     T4207
      ORB
      OR      M4209  ; 2P INFRA AUTO END
      ANI     T4209  ; 2P INFRA AUTO END
      OUT     M4209  ; 2P INFRA AUTO END
      OUT     T4209 K1  ; 2P INFRA AUTO END
; [Title]2P INFRA WLED FRONT (6 POINT)
; INFRA 2P WELD FRONT #1
2773  LDI     SM400  ; ALWAYS ON
      ORP     B11  ; 임시AT.2P.FRONT.#1
      LD      B1061  ; MODEL#1.2P 18S-S
      OR      B1062  ; MODEL#2.2P 18S-R
      AND     M4106  ; 2P INFRA WELDING START
      ORB
      OR      M4110  ; INFRA.2P.FR.#1.AT
      ANI     T4116
      OUT     M4110  ; INFRA.2P.FR.#1.AT
      OUT     T4110 K1
